LIN {X 0,Y 119.711,Z 958.893,A -85,B 0,C 180,E1 26114.773,E2 26114.773} C_VEL
LIN {X 0,Y 103.923,Z 964.098,A -85,B 0,C 180,E1 26117.575,E2 26117.575} C_VEL
LIN {X 0,Y 73.939,Z 972.907,A -85,B 0,C 180,E1 26135.275,E2 26135.275} C_VEL
LIN {X 0,Y 58.903,Z 976.31,A -85,B 0,C 180,E1 26159.176,E2 26159.176} C_VEL
LIN {X 0,Y 56.099,Z 976.57,A -85,B 0,C 180,E1 26189.998,E2 26189.998} C_VEL
LIN {X 0,Y 59.186,Z 972.492,A -85,B 0,C 180,E1 26220.657,E2 26220.657} C_VEL
LIN {X 0,Y 76.443,Z 963.091,A -85,B 0,C 180,E1 26247.029,E2 26247.029} C_VEL
LIN {X 0,Y 104.465,Z 947.144,A -85,B 0,C 180,E1 26263.142,E2 26263.142} C_VEL
LIN {X 0,Y 134.627,Z 925.946,A -85,B 0,C 180,E1 26271.712,E2 26271.712} C_VEL
LIN {X 0,Y 162.508,Z 900.972,A -85,B 0,C 180,E1 26276.579,E2 26276.579} C_VEL
LIN {X 0,Y 170.712,Z 892.031,A -85,B 0,C 180,E1 26277.998,E2 26277.998} C_VEL
LIN {X 0,Y 172.966,Z 882.755,A -85,B 0,C 180,E1 26286.219,E2 26286.219} C_VEL
LIN {X 0,Y 173.334,Z 880.134,A -85,B 0,C 180,E1 26289.984,E2 26289.984} C_VEL
LIN {X 0,Y 171.958,Z 879.719,A -85,B 0,C 180,E1 26295.218,E2 26295.218} C_VEL
LIN {X 0,Y 170.223,Z 881.343,A -85,B 0,C 180,E1 26303.461,E2 26303.461} C_VEL
LIN {X 0,Y 168.527,Z 885.017,A -85,B 0,C 180,E1 26309.922,E2 26309.922} C_VEL
LIN {X 0,Y 166.252,Z 890.112,A -85,B 0,C 180,E1 26315.225,E2 26315.225} C_VEL
LIN {X 0,Y 138.554,Z 915.597,A -85,B 0,C 180,E1 26320.326,E2 26320.326} C_VEL
LIN {X 0,Y 110.78,Z 935.517,A -85,B 0,C 180,E1 26327.957,E2 26327.957} C_VEL
LIN {X 0,Y 84.761,Z 950.496,A -85,B 0,C 180,E1 26340.688,E2 26340.688} C_VEL
LIN {X 0,Y 63.942,Z 960.925,A -85,B 0,C 180,E1 26363.225,E2 26363.225} C_VEL
LIN {X 0,Y 56.022,Z 965.379,A -85,B 0,C 180,E1 26385.628,E2 26385.628} C_VEL
LIN {X 0,Y 59.105,Z 968.135,A -85,B 0,C 180,E1 26419.994,E2 26419.994} C_VEL
LIN {X 0,Y 77.778,Z 966.879,A -85,B 0,C 180,E1 26445.956,E2 26445.956} C_VEL
LIN {X 0,Y 110.4,Z 960.103,A -85,B 0,C 180,E1 26463.301,E2 26463.301} C_VEL
LIN {X 0,Y 132.48,Z 953.174,A -85,B 0,C 180,E1 26469.432,E2 26469.432} C_VEL
LIN {X 0,Y 103.923,Z 964.098,A -85,B 0,C 180,E1 26477.575,E2 26477.575} C_VEL
LIN {X 0,Y 88.187,Z 968.35,A -85,B 0,C 180,E1 26481.478,E2 26481.478} C_VEL
LIN {X 0,Y 72.86,Z 971.58,A -85,B 0,C 180,E1 26487.114,E2 26487.114} C_VEL
LIN {X 0,Y 52.121,Z 975.608,A -85,B 0,C 180,E1 26514.614,E2 26514.614} C_VEL
LIN {X 0,Y 48.161,Z 975.76,A -85,B 0,C 180,E1 26549.998,E2 26549.998} C_VEL
LIN {X 0,Y 52.398,Z 971.472,A -85,B 0,C 180,E1 26585.166,E2 26585.166} C_VEL
LIN {X 0,Y 72.034,Z 961.958,A -85,B 0,C 180,E1 26612.291,E2 26612.291} C_VEL
LIN {X 0,Y 102.362,Z 945.563,A -85,B 0,C 180,E1 26627.605,E2 26627.605} C_VEL
LIN {X 0,Y 132.171,Z 925.212,A -85,B 0,C 180,E1 26634.962,E2 26634.962} C_VEL
LIN {X 0,Y 161.894,Z 898.969,A -85,B 0,C 180,E1 26639.462,E2 26639.462} C_VEL
LIN {X 0,Y 165.333,Z 895.412,A -85,B 0,C 180,E1 26639.958,E2 26639.958} C_VEL
LIN {X 0,Y 167.77,Z 887.011,A -85,B 0,C 180,E1 26648.352,E2 26648.352} C_VEL
LIN {X 0,Y 167.887,Z 885.942,A -85,B 0,C 180,E1 26650.312,E2 26650.312} C_VEL
LIN {X 0,Y 166.423,Z 885.651,A -85,B 0,C 180,E1 26655.737,E2 26655.737} C_VEL
LIN {X 0,Y 164.66,Z 887.179,A -85,B 0,C 180,E1 26663.589,E2 26663.589} C_VEL
LIN {X 0,Y 163.034,Z 890.313,A -85,B 0,C 180,E1 26669.203,E2 26669.203} C_VEL
LIN {X 0,Y 161.386,Z 893.294,A -85,B 0,C 180,E1 26672.698,E2 26672.698} C_VEL
LIN {X 0,Y 152.966,Z 901.547,A -85,B 0,C 180,E1 26674.291,E2 26674.291} C_VEL
LIN {X 0,Y 123.005,Z 925.698,A -85,B 0,C 180,E1 26679.938,E2 26679.938} C_VEL
LIN {X 0,Y 92.965,Z 944.319,A -85,B 0,C 180,E1 26689.514,E2 26689.514} C_VEL
LIN {X 0,Y 66.823,Z 957.209,A -85,B 0,C 180,E1 26706.828,E2 26706.828} C_VEL
LIN {X 0,Y 52.071,Z 963.832,A -85,B 0,C 180,E1 26730.002,E2 26730.002} C_VEL
LIN {X 0,Y 48.032,Z 968.202,A -85,B 0,C 180,E1 26768.931,E2 26768.931} C_VEL
LIN {X 0,Y 63.418,Z 968.657,A -85,B 0,C 180,E1 26802.143,E2 26802.143} C_VEL
LIN {X 0,Y 96.013,Z 964.023,A -85,B 0,C 180,E1 26823.196,E2 26823.196} C_VEL
LIN {X 0,Y 114.587,Z 959.44,A -85,B 0,C 180,E1 26829.148,E2 26829.148} C_VEL
LIN {X 0,Y 80.764,Z 969.716,A -85,B 0,C 180,E1 26842.03,E2 26842.03} C_VEL
LIN {X 0,Y 72.86,Z 971.58,A -85,B 0,C 180,E1 26847.114,E2 26847.114} C_VEL
LIN {X 0,Y 58.467,Z 973.826,A -85,B 0,C 180,E1 26855.615,E2 26855.615} C_VEL
LIN {X 0,Y 45.635,Z 974.913,A -85,B 0,C 180,E1 26868.941,E2 26868.941} C_VEL
LIN {X 0,Y 40.215,Z 974.944,A -85,B 0,C 180,E1 26909.997,E2 26909.997} C_VEL
LIN {X 0,Y 45.994,Z 970.426,A -85,B 0,C 180,E1 26951.006,E2 26951.006} C_VEL
LIN {X 0,Y 71.033,Z 959.531,A -85,B 0,C 180,E1 26979.966,E2 26979.966} C_VEL
LIN {X 0,Y 100.479,Z 944.235,A -85,B 0,C 180,E1 26992.068,E2 26992.068} C_VEL
LIN {X 0,Y 132.074,Z 922.944,A -85,B 0,C 180,E1 26998.663,E2 26998.663} C_VEL
LIN {X 0,Y 160.083,Z 898.33,A -85,B 0,C 180,E1 27002.382,E2 27002.382} C_VEL
LIN {X 0,Y 162.144,Z 892.536,A -85,B 0,C 180,E1 27008.644,E2 27008.644} C_VEL
LIN {X 0,Y 162.183,Z 891.558,A -85,B 0,C 180,E1 27010.679,E2 27010.679} C_VEL
LIN {X 0,Y 159.928,Z 891.844,A -85,B 0,C 180,E1 27019.343,E2 27019.343} C_VEL
LIN {X 0,Y 158.168,Z 894.158,A -85,B 0,C 180,E1 27026.512,E2 27026.512} C_VEL
LIN {X 0,Y 155.869,Z 897.582,A -85,B 0,C 180,E1 27030.772,E2 27030.772} C_VEL
LIN {X 0,Y 125.105,Z 922.932,A -85,B 0,C 180,E1 27035.494,E2 27035.494} C_VEL
LIN {X 0,Y 93.629,Z 942.489,A -85,B 0,C 180,E1 27043.511,E2 27043.511} C_VEL
LIN {X 0,Y 65.062,Z 956.148,A -85,B 0,C 180,E1 27058.545,E2 27058.545} C_VEL
LIN {X 0,Y 45.303,Z 964.232,A -85,B 0,C 180,E1 27085.116,E2 27085.116} C_VEL
LIN {X 0,Y 41.415,Z 969.099,A -85,B 0,C 180,E1 27136.784,E2 27136.784} C_VEL
LIN {X 0,Y 61.198,Z 969.344,A -85,B 0,C 180,E1 27170.523,E2 27170.523} C_VEL
LIN {X 0,Y 97.33,Z 964.29,A -85,B 0,C 180,E1 27188.989,E2 27188.989} C_VEL
LIN {X 0,Y 65.834,Z 971.78,A -85,B 0,C 180,E1 27203.524,E2 27203.524} C_VEL
LIN {X 0,Y 45.635,Z 974.913,A -85,B 0,C 180,E1 27228.941,E2 27228.941} C_VEL
LIN {X 0,Y 36.743,Z 974.992,A -85,B 0,C 180,E1 27250.159,E2 27250.159} C_VEL
LIN {X 0,Y 31.959,Z 973.487,A -85,B 0,C 180,E1 27279.171,E2 27279.171} C_VEL
LIN {X 0,Y 40.22,Z 969.374,A -85,B 0,C 180,E1 27318.619,E2 27318.619} C_VEL
LIN {X 0,Y 66.986,Z 958.913,A -85,B 0,C 180,E1 27345.601,E2 27345.601} C_VEL
LIN {X 0,Y 100.621,Z 942.076,A -85,B 0,C 180,E1 27356.978,E2 27356.978} C_VEL
LIN {X 0,Y 134.05,Z 919.516,A -85,B 0,C 180,E1 27362.481,E2 27362.481} C_VEL
LIN {X 0,Y 154.859,Z 901.45,A -85,B 0,C 180,E1 27364.846,E2 27364.846} C_VEL
LIN {X 0,Y 156.143,Z 898.412,A -85,B 0,C 180,E1 27368.288,E2 27368.288} C_VEL
LIN {X 0,Y 156.339,Z 897.044,A -85,B 0,C 180,E1 27371.083,E2 27371.083} C_VEL
LIN {X 0,Y 154.75,Z 897.004,A -85,B 0,C 180,E1 27376.959,E2 27376.959} C_VEL
LIN {X 0,Y 153.208,Z 898.276,A -85,B 0,C 180,E1 27383.147,E2 27383.147} C_VEL
LIN {X 0,Y 151.455,Z 900.693,A -85,B 0,C 180,E1 27388.014,E2 27388.014} C_VEL
LIN {X 0,Y 122.429,Z 923.851,A -85,B 0,C 180,E1 27392.072,E2 27392.072} C_VEL
LIN {X 0,Y 91.761,Z 942.438,A -85,B 0,C 180,E1 27398.636,E2 27398.636} C_VEL
LIN {X 0,Y 61.36,Z 956.339,A -85,B 0,C 180,E1 27412.063,E2 27412.063} C_VEL
LIN {X 0,Y 37.169,Z 965.222,A -85,B 0,C 180,E1 27442.856,E2 27442.856} C_VEL
LIN {X 0,Y 31.309,Z 968.568,A -85,B 0,C 180,E1 27478.818,E2 27478.818} C_VEL
LIN {X 0,Y 46.446,Z 970.459,A -85,B 0,C 180,E1 27527.092,E2 27527.092} C_VEL
LIN {X 0,Y 80.023,Z 967.951,A -85,B 0,C 180,E1 27548.91,E2 27548.91} C_VEL
LIN {X 0,Y 50.488,Z 973.087,A -85,B 0,C 180,E1 27566.272,E2 27566.272} C_VEL
LIN {X 0,Y 32.535,Z 974.518,A -85,B 0,C 180,E1 27608.614,E2 27608.614} C_VEL
LIN {X 0,Y 32.289,Z 974.094,A -85,B 0,C 180,E1 27629.997,E2 27629.997} C_VEL
LIN {X 0,Y 31.959,Z 973.487,A -85,B 0,C 180,E1 27639.171,E2 27639.171} C_VEL
LIN {X 0,Y 31.956,Z 971.586,A -85,B 0,C 180,E1 27662.601,E2 27662.601} C_VEL
LIN {X 0,Y 40.054,Z 966.811,A -85,B 0,C 180,E1 27695.217,E2 27695.217} C_VEL
LIN {X 0,Y 72.676,Z 954.478,A -85,B 0,C 180,E1 27715.255,E2 27715.255} C_VEL
LIN {X 0,Y 105.736,Z 937.275,A -85,B 0,C 180,E1 27722.569,E2 27722.569} C_VEL
LIN {X 0,Y 138.365,Z 914.337,A -85,B 0,C 180,E1 27726.394,E2 27726.394} C_VEL
LIN {X 0,Y 148.68,Z 905.586,A -85,B 0,C 180,E1 27727.21,E2 27727.21} C_VEL
LIN {X 0,Y 150.135,Z 903.774,A -85,B 0,C 180,E1 27728.542,E2 27728.542} C_VEL
LIN {X 0,Y 150.356,Z 902.432,A -85,B 0,C 180,E1 27731.53,E2 27731.53} C_VEL
LIN {X 0,Y 147.324,Z 903.497,A -85,B 0,C 180,E1 27742.802,E2 27742.802} C_VEL
LIN {X 0,Y 145.718,Z 905.164,A -85,B 0,C 180,E1 27745.71,E2 27745.71} C_VEL
LIN {X 0,Y 112.822,Z 929.64,A -85,B 0,C 180,E1 27749.614,E2 27749.614} C_VEL
LIN {X 0,Y 79.724,Z 947.662,A -85,B 0,C 180,E1 27756.446,E2 27756.446} C_VEL
LIN {X 0,Y 48.468,Z 960.086,A -85,B 0,C 180,E1 27771.491,E2 27771.491} C_VEL
LIN {X 0,Y 26.098,Z 967.262,A -85,B 0,C 180,E1 27810.004,E2 27810.004} C_VEL
LIN {X 0,Y 31.853,Z 970.838,A -85,B 0,C 180,E1 27881.359,E2 27881.359} C_VEL
LIN {X 0,Y 61.018,Z 970.628,A -85,B 0,C 180,E1 27908.402,E2 27908.402} C_VEL
LIN {X 0,Y 61.163,Z 970.689,A -85,B 0,C 180,E1 27909.277,E2 27909.277} C_VEL
LIN {X 0,Y 35.19,Z 973.51,A -85,B 0,C 180,E1 27930.941,E2 27930.941} C_VEL
LIN {X 0,Y 24.337,Z 973.195,A -85,B 0,C 180,E1 27989.995,E2 27989.995} C_VEL
LIN {X 0,Y 35.366,Z 968.304,A -85,B 0,C 180,E1 28048.575,E2 28048.575} C_VEL
LIN {X 0,Y 40.054,Z 966.811,A -85,B 0,C 180,E1 28055.217,E2 28055.217} C_VEL
LIN {X 0,Y 46.016,Z 964.52,A -85,B 0,C 180,E1 28063.199,E2 28063.199} C_VEL
LIN {X 0,Y 63.342,Z 956.829,A -85,B 0,C 180,E1 28079.399,E2 28079.399} C_VEL
LIN {X 0,Y 65.271,Z 956.031,A -85,B 0,C 180,E1 28080.019,E2 28080.019} C_VEL
LIN {X 0,Y 100.591,Z 938.959,A -85,B 0,C 180,E1 28086.367,E2 28086.367} C_VEL
LIN {X 0,Y 133.651,Z 916.81,A -85,B 0,C 180,E1 28089.355,E2 28089.355} C_VEL
LIN {X 0,Y 144.15,Z 908.185,A -85,B 0,C 180,E1 28090.179,E2 28090.179} C_VEL
LIN {X 0,Y 142.563,Z 907.744,A -85,B 0,C 180,E1 28097.705,E2 28097.705} C_VEL
LIN {X 0,Y 140.416,Z 909.376,A -85,B 0,C 180,E1 28102.97,E2 28102.97} C_VEL
LIN {X 0,Y 107.202,Z 932.703,A -85,B 0,C 180,E1 28106.187,E2 28106.187} C_VEL
LIN {X 0,Y 75.19,Z 949.25,A -85,B 0,C 180,E1 28111.469,E2 28111.469} C_VEL
LIN {X 0,Y 42.298,Z 961.373,A -85,B 0,C 180,E1 28124.481,E2 28124.481} C_VEL
LIN {X 0,Y 17.317,Z 968.386,A -85,B 0,C 180,E1 28170.007,E2 28170.007} C_VEL
LIN {X 0,Y 32.04,Z 971.828,A -85,B 0,C 180,E1 28260.217,E2 28260.217} C_VEL
LIN {X 0,Y 42.169,Z 972.094,A -85,B 0,C 180,E1 28269.553,E2 28269.553} C_VEL
LIN {X 0,Y 16.495,Z 972.674,A -85,B 0,C 180,E1 28327.215,E2 28327.215} C_VEL
LIN {X 0,Y 16.391,Z 972.293,A -85,B 0,C 180,E1 28349.993,E2 28349.993} C_VEL
LIN {X 0,Y 31.887,Z 967.221,A -85,B 0,C 180,E1 28421.159,E2 28421.159} C_VEL
LIN {X 0,Y 65.271,Z 956.031,A -85,B 0,C 180,E1 28440.019,E2 28440.019} C_VEL
LIN {X 0,Y 79.491,Z 949.248,A -85,B 0,C 180,E1 28446.128,E2 28446.128} C_VEL
LIN {X 0,Y 93.92,Z 941.499,A -85,B 0,C 180,E1 28450.39,E2 28450.39} C_VEL
LIN {X 0,Y 127.879,Z 920.126,A -85,B 0,C 180,E1 28452.538,E2 28452.538} C_VEL
LIN {X 0,Y 136.131,Z 913.817,A -85,B 0,C 180,E1 28452.903,E2 28452.903} C_VEL
LIN {X 0,Y 137.462,Z 912.657,A -85,B 0,C 180,E1 28453.417,E2 28453.417} C_VEL
LIN {X 0,Y 135.813,Z 913.036,A -85,B 0,C 180,E1 28459.412,E2 28459.412} C_VEL
LIN {X 0,Y 134.055,Z 914.378,A -85,B 0,C 180,E1 28460.104,E2 28460.104} C_VEL
LIN {X 0,Y 100.047,Z 936.867,A -85,B 0,C 180,E1 28462.509,E2 28462.509} C_VEL
LIN {X 0,Y 63.663,Z 953.883,A -85,B 0,C 180,E1 28467.257,E2 28467.257} C_VEL
LIN {X 0,Y 29.277,Z 964.672,A -85,B 0,C 180,E1 28479.369,E2 28479.369} C_VEL
LIN {X 0,Y 7.722,Z 970.149,A -85,B 0,C 180,E1 28568.263,E2 28568.263} C_VEL
LIN {X 0,Y 21.172,Z 972.047,A -85,B 0,C 180,E1 28627.608,E2 28627.608} C_VEL
LIN {X 0,Y 16.058,Z 972.08,A -85,B 0,C 180,E1 28639.974,E2 28639.974} C_VEL
LIN {X 0,Y 8.431,Z 971.381,A -85,B 0,C 180,E1 28709.987,E2 28709.987} C_VEL
LIN {X 0,Y 30.254,Z 966.123,A -85,B 0,C 180,E1 28795.944,E2 28795.944} C_VEL
LIN {X 0,Y 68.056,Z 953.688,A -85,B 0,C 180,E1 28807.554,E2 28807.554} C_VEL
LIN {X 0,Y 93.92,Z 941.499,A -85,B 0,C 180,E1 28810.39,E2 28810.39} C_VEL
LIN {X 0,Y 108.248,Z 933.006,A -85,B 0,C 180,E1 28813.505,E2 28813.505} C_VEL
LIN {X 0,Y 122.196,Z 923.511,A -85,B 0,C 180,E1 28815.958,E2 28815.958} C_VEL
LIN {X 0,Y 129.102,Z 918.581,A -85,B 0,C 180,E1 28816.078,E2 28816.078} C_VEL
LIN {X 0,Y 124.315,Z 921.857,A -85,B 0,C 180,E1 28816.988,E2 28816.988} C_VEL
LIN {X 0,Y 90.831,Z 942.024,A -85,B 0,C 180,E1 28818.318,E2 28818.318} C_VEL
LIN {X 0,Y 52.563,Z 958.116,A -85,B 0,C 180,E1 28821.092,E2 28821.092} C_VEL
LIN {X 0,Y 24.778,Z 965.851,A -85,B 0,C 180,E1 28824.015,E2 28824.015} C_VEL
LIN {X 0,Y 0.464,Z 970.462,A -85,B 0,C 180,E1 28709.757,E2 28709.757} C_VEL
LIN {X 0,Y 30.769,Z 964.938,A -85,B 0,C 180,E1 28811.24,E2 28811.24} C_VEL
LIN {X 0,Y 66.139,Z 953.616,A -85,B 0,C 180,E1 28814.152,E2 28814.152} C_VEL
LIN {X 0,Y 101.772,Z 936.397,A -85,B 0,C 180,E1 28815.471,E2 28815.471} C_VEL
LIN {X 0,Y 122.196,Z 923.511,A -85,B 0,C 180,E1 28815.958,E2 28815.958} C_VEL
LIN {X 0,Y 125.353,Z 925.139,A -85,B 0,C 180,E1 28816.04,E2 28816.04} C_VEL
LIN {X 0,Y 125.353,Z 1015.5,A -85,B 0,C 180,E1 28816.04,E2 28816.04} C_VEL
LIN {X 0,Y 125.353,Z 1015.5,A -85,B 0,C 180,E1 28816.04,E2 28816.04}

QRS_NEXT_CUT()
PTP {E1 28976.873,E2 28976.873}
PTP {X 0,Y 607.916,A -85,B 0,C 180,E1 28976.873,E2 28976.873,E3 0,E4 0,E5 0,E6 0}
QRS_SPEED_INIT()
LIN {X 0,Y 607.916,Z 1015.5,A -85,B 0,C 180,E1 28976.873,E2 28976.873,E3 0,E4 0,E5 0,E6 0} C_VEL
LIN {X 0,Y 607.916,Z 400.085,A -85,B 0,C 180,E1 28976.873,E2 28976.873} C_VEL
LIN {X 0,Y 607.916,Z 392.009,A -85,B 0,C 180,E1 28976.873,E2 28976.873} C_VEL
LIN {X 0,Y 607.891,Z 390.009,A -85,B 0,C 180,E1 28976.684,E2 28976.684} C_VEL
LIN {X 0,Y 607.87,Z 390.013,A -85,B 0,C 180,E1 28973.673,E2 28973.673} C_VEL
LIN {X 0,Y 607.89,Z 390.008,A -85,B 0,C 180,E1 28970.437,E2 28970.437} C_VEL
LIN {X 0,Y 607.892,Z 390.014,A -85,B 0,C 180,E1 28967.364,E2 28967.364} C_VEL
LIN {X 0,Y 607.887,Z 390.007,A -85,B 0,C 180,E1 28964.155,E2 28964.155} C_VEL
LIN {X 0,Y 607.914,Z 390.015,A -85,B 0,C 180,E1 28960.994,E2 28960.994} C_VEL
LIN {X 0,Y 607.883,Z 390.008,A -85,B 0,C 180,E1 28957.771,E2 28957.771} C_VEL
LIN {X 0,Y 607.906,Z 390.012,A -85,B 0,C 180,E1 28954.682,E2 28954.682} C_VEL
LIN {X 0,Y 607.888,Z 390.01,A -85,B 0,C 180,E1 28951.51,E2 28951.51} C_VEL
LIN {X 0,Y 607.904,Z 390.198,A -85,B 0,C 180,E1 28949.07,E2 28949.07} C_VEL
LIN {X 0,Y 607.917,Z 394.228,A -85,B 0,C 180,E1 28948.733,E2 28948.733} C_VEL
LIN {X 0,Y 607.919,Z 437.692,A -85,B 0,C 180,E1 28945.648,E2 28945.648} C_VEL
LIN {X 0,Y 607.909,Z 452.342,A -85,B 0,C 180,E1 28944.642,E2 28944.642} C_VEL
LIN {X 0,Y 607.915,Z 681.342,A -85,B 0,C 180,E1 28941.679,E2 28941.679} C_VEL
LIN {X 0,Y 607.916,Z 715.007,A -85,B 0,C 180,E1 28941.219,E2 28941.219} C_VEL
LIN {X 0,Y 607.906,Z 735.187,A -85,B 0,C 180,E1 28940.771,E2 28940.771} C_VEL
LIN {X 0,Y 607.911,Z 754.308,A -85,B 0,C 180,E1 28940.178,E2 28940.178} C_VEL
LIN {X 0,Y 607.909,Z 774.728,A -85,B 0,C 180,E1 28939.358,E2 28939.358} C_VEL
LIN {X 0,Y 607.917,Z 793.066,A -85,B 0,C 180,E1 28938.443,E2 28938.443} C_VEL
LIN {X 0,Y 607.916,Z 811.339,A -85,B 0,C 180,E1 28937.341,E2 28937.341} C_VEL
LIN {X 0,Y 607.914,Z 829.252,A -85,B 0,C 180,E1 28936.046,E2 28936.046} C_VEL
LIN {X 0,Y 607.917,Z 846.214,A -85,B 0,C 180,E1 28934.588,E2 28934.588} C_VEL
LIN {X 0,Y 607.909,Z 861.448,A -85,B 0,C 180,E1 28933.04,E2 28933.04} C_VEL
LIN {X 0,Y 607.918,Z 875.235,A -85,B 0,C 180,E1 28931.386,E2 28931.386} C_VEL
LIN {X 0,Y 607.914,Z 887.272,A -85,B 0,C 180,E1 28929.669,E2 28929.669} C_VEL
LIN {X 0,Y 607.905,Z 897.319,A -85,B 0,C 180,E1 28927.958,E2 28927.958} C_VEL
LIN {X 0,Y 607.901,Z 906.432,A -85,B 0,C 180,E1 28926.07,E2 28926.07} C_VEL
LIN {X 0,Y 607.9,Z 913.506,A -85,B 0,C 180,E1 28924.226,E2 28924.226} C_VEL
LIN {X 0,Y 607.899,Z 919.069,A -85,B 0,C 180,E1 28922.31,E2 28922.31} C_VEL
LIN {X 0,Y 607.9,Z 922.757,A -85,B 0,C 180,E1 28920.434,E2 28920.434} C_VEL
LIN {X 0,Y 607.9,Z 924.923,A -85,B 0,C 180,E1 28918.485,E2 28918.485} C_VEL
LIN {X 0,Y 607.902,Z 925.392,A -85,B 0,C 180,E1 28916.467,E2 28916.467} C_VEL
LIN {X 0,Y 607.907,Z 924.09,A -85,B 0,C 180,E1 28914.483,E2 28914.483} C_VEL
LIN {X 0,Y 607.914,Z 921.318,A -85,B 0,C 180,E1 28912.633,E2 28912.633} C_VEL
LIN {X 0,Y 607.918,Z 916.682,A -85,B 0,C 180,E1 28910.706,E2 28910.706} C_VEL
LIN {X 0,Y 607.909,Z 910.708,A -85,B 0,C 180,E1 28908.903,E2 28908.903} C_VEL
LIN {X 0,Y 607.9,Z 902.729,A -85,B 0,C 180,E1 28907.021,E2 28907.021} C_VEL
LIN {X 0,Y 607.903,Z 893.474,A -85,B 0,C 180,E1 28905.255,E2 28905.255} C_VEL
LIN {X 0,Y 607.907,Z 882.395,A -85,B 0,C 180,E1 28903.504,E2 28903.504} C_VEL
LIN {X 0,Y 607.913,Z 869.197,A -85,B 0,C 180,E1 28901.765,E2 28901.765} C_VEL
LIN {X 0,Y 607.914,Z 854.508,A -85,B 0,C 180,E1 28900.134,E2 28900.134} C_VEL
LIN {X 0,Y 607.916,Z 838.768,A -85,B 0,C 180,E1 28898.653,E2 28898.653} C_VEL
LIN {X 0,Y 607.915,Z 822.476,A -85,B 0,C 180,E1 28897.352,E2 28897.352} C_VEL
LIN {X 0,Y 607.918,Z 805.221,A -85,B 0,C 180,E1 28896.182,E2 28896.182} C_VEL
LIN {X 0,Y 607.916,Z 786.897,A -85,B 0,C 180,E1 28895.141,E2 28895.141} C_VEL
LIN {X 0,Y 607.917,Z 768.828,A -85,B 0,C 180,E1 28894.29,E2 28894.29} C_VEL
LIN {X 0,Y 607.916,Z 749.3,A -85,B 0,C 180,E1 28893.558,E2 28893.558} C_VEL
LIN {X 0,Y 607.908,Z 730.169,A -85,B 0,C 180,E1 28893.015,E2 28893.015} C_VEL
LIN {X 0,Y 607.912,Z 709.347,A -85,B 0,C 180,E1 28892.602,E2 28892.602} C_VEL
LIN {X 0,Y 607.91,Z 453.431,A -85,B 0,C 180,E1 28889.291,E2 28889.291} C_VEL
LIN {X 0,Y 607.904,Z 451.144,A -85,B 0,C 180,E1 28889.197,E2 28889.197} C_VEL
LIN {X 0,Y 607.918,Z 406.873,A -85,B 0,C 180,E1 28886.084,E2 28886.084} C_VEL
LIN {X 0,Y 607.905,Z 390.386,A -85,B 0,C 180,E1 28884.879,E2 28884.879} C_VEL
LIN {X 0,Y 607.885,Z 390.007,A -85,B 0,C 180,E1 28884.334,E2 28884.334} C_VEL
LIN {X 0,Y 607.904,Z 390.011,A -85,B 0,C 180,E1 28881.2,E2 28881.2} C_VEL
LIN {X 0,Y 607.888,Z 390.007,A -85,B 0,C 180,E1 28878.037,E2 28878.037} C_VEL
LIN {X 0,Y 607.906,Z 390.012,A -85,B 0,C 180,E1 28874.901,E2 28874.901} C_VEL
LIN {X 0,Y 607.89,Z 390.007,A -85,B 0,C 180,E1 28871.788,E2 28871.788} C_VEL
LIN {X 0,Y 607.909,Z 390.013,A -85,B 0,C 180,E1 28868.581,E2 28868.581} C_VEL
LIN {X 0,Y 607.905,Z 390.004,A -85,B 0,C 180,E1 28865.305,E2 28865.305} C_VEL
LIN {X 0,Y 607.905,Z 390.013,A -85,B 0,C 180,E1 28862.036,E2 28862.036} C_VEL
LIN {X 0,Y 607.908,Z 390.005,A -85,B 0,C 180,E1 28858.79,E2 28858.79} C_VEL
LIN {X 0,Y 607.895,Z 390.011,A -85,B 0,C 180,E1 28855.655,E2 28855.655} C_VEL
LIN {X 0,Y 607.904,Z 390.006,A -85,B 0,C 180,E1 28852.513,E2 28852.513} C_VEL
LIN {X 0,Y 607.892,Z 390.01,A -85,B 0,C 180,E1 28849.311,E2 28849.311} C_VEL
LIN {X 0,Y 607.9,Z 390.007,A -85,B 0,C 180,E1 28846.175,E2 28846.175} C_VEL
LIN {X 0,Y 607.892,Z 390.009,A -85,B 0,C 180,E1 28843.047,E2 28843.047} C_VEL
LIN {X 0,Y 607.898,Z 390.008,A -85,B 0,C 180,E1 28839.901,E2 28839.901} C_VEL
LIN {X 0,Y 607.892,Z 390.008,A -85,B 0,C 180,E1 28836.772,E2 28836.772} C_VEL
LIN {X 0,Y 607.896,Z 390.009,A -85,B 0,C 180,E1 28833.662,E2 28833.662} C_VEL
LIN {X 0,Y 607.893,Z 390.009,A -85,B 0,C 180,E1 28830.547,E2 28830.547} C_VEL
LIN {X 0,Y 607.897,Z 390.009,A -85,B 0,C 180,E1 28827.422,E2 28827.422} C_VEL
LIN {X 0,Y 607.893,Z 390.008,A -85,B 0,C 180,E1 28824.28,E2 28824.28} C_VEL
LIN {X 0,Y 607.897,Z 390.01,A -85,B 0,C 180,E1 28821.113,E2 28821.113} C_VEL
LIN {X 0,Y 607.896,Z 390.008,A -85,B 0,C 180,E1 28818.013,E2 28818.013} C_VEL
LIN {X 0,Y 607.896,Z 390.01,A -85,B 0,C 180,E1 28814.868,E2 28814.868} C_VEL
LIN {X 0,Y 607.9,Z 390.006,A -85,B 0,C 180,E1 28811.672,E2 28811.672} C_VEL
LIN {X 0,Y 607.901,Z 390.011,A -85,B 0,C 180,E1 28808.513,E2 28808.513} C_VEL
LIN {X 0,Y 607.911,Z 390.004,A -85,B 0,C 180,E1 28805.285,E2 28805.285} C_VEL
LIN {X 0,Y 607.912,Z 390.015,A -85,B 0,C 180,E1 28801.98,E2 28801.98} C_VEL
LIN {X 0,Y 607.899,Z 390.006,A -85,B 0,C 180,E1 28798.681,E2 28798.681} C_VEL
LIN {X 0,Y 607.9,Z 390.011,A -85,B 0,C 180,E1 28795.472,E2 28795.472} C_VEL
LIN {X 0,Y 607.893,Z 390.007,A -85,B 0,C 180,E1 28792.344,E2 28792.344} C_VEL
LIN {X 0,Y 607.899,Z 390.01,A -85,B 0,C 180,E1 28789.193,E2 28789.193} C_VEL
LIN {X 0,Y 607.892,Z 390.007,A -85,B 0,C 180,E1 28786.105,E2 28786.105} C_VEL
LIN {X 0,Y 607.9,Z 390.01,A -85,B 0,C 180,E1 28782.976,E2 28782.976} C_VEL
LIN {X 0,Y 607.891,Z 390.007,A -85,B 0,C 180,E1 28779.894,E2 28779.894} C_VEL
LIN {X 0,Y 607.901,Z 390.01,A -85,B 0,C 180,E1 28776.75,E2 28776.75} C_VEL
LIN {X 0,Y 607.889,Z 390.008,A -85,B 0,C 180,E1 28773.635,E2 28773.635} C_VEL
LIN {X 0,Y 607.901,Z 390.01,A -85,B 0,C 180,E1 28770.542,E2 28770.542} C_VEL
LIN {X 0,Y 607.889,Z 390.007,A -85,B 0,C 180,E1 28767.463,E2 28767.463} C_VEL
LIN {X 0,Y 607.903,Z 390.01,A -85,B 0,C 180,E1 28764.343,E2 28764.343} C_VEL
LIN {X 0,Y 607.887,Z 390.008,A -85,B 0,C 180,E1 28761.195,E2 28761.195} C_VEL
LIN {X 0,Y 607.903,Z 390.01,A -85,B 0,C 180,E1 28758.105,E2 28758.105} C_VEL
LIN {X 0,Y 607.887,Z 390.008,A -85,B 0,C 180,E1 28754.987,E2 28754.987} C_VEL
LIN {X 0,Y 607.902,Z 390.01,A -85,B 0,C 180,E1 28751.897,E2 28751.897} C_VEL
LIN {X 0,Y 607.886,Z 390.008,A -85,B 0,C 180,E1 28748.773,E2 28748.773} C_VEL
LIN {X 0,Y 607.899,Z 390.272,A -85,B 0,C 180,E1 28746.232,E2 28746.232} C_VEL
LIN {X 0,Y 607.915,Z 394.031,A -85,B 0,C 180,E1 28745.958,E2 28745.958} C_VEL
LIN {X 0,Y 607.913,Z 445.359,A -85,B 0,C 180,E1 28742.929,E2 28742.929} C_VEL
LIN {X 0,Y 607.903,Z 455.392,A -85,B 0,C 180,E1 28742.37,E2 28742.37} C_VEL
LIN {X 0,Y 607.916,Z 672.013,A -85,B 0,C 180,E1 28739.445,E2 28739.445} C_VEL
LIN {X 0,Y 607.899,Z 760.574,A -85,B 0,C 180,E1 28738.249,E2 28738.249} C_VEL
LIN {X 0,Y 607.906,Z 781.2,A -85,B 0,C 180,E1 28737.806,E2 28737.806} C_VEL
LIN {X 0,Y 607.908,Z 801.762,A -85,B 0,C 180,E1 28737.211,E2 28737.211} C_VEL
LIN {X 0,Y 607.904,Z 822.538,A -85,B 0,C 180,E1 28736.419,E2 28736.419} C_VEL
LIN {X 0,Y 607.918,Z 843.715,A -85,B 0,C 180,E1 28735.423,E2 28735.423} C_VEL
LIN {X 0,Y 607.916,Z 863.098,A -85,B 0,C 180,E1 28734.332,E2 28734.332} C_VEL
LIN {X 0,Y 607.915,Z 881.539,A -85,B 0,C 180,E1 28733.097,E2 28733.097} C_VEL
LIN {X 0,Y 607.911,Z 899.771,A -85,B 0,C 180,E1 28731.678,E2 28731.678} C_VEL
LIN {X 0,Y 607.913,Z 916.635,A -85,B 0,C 180,E1 28730.157,E2 28730.157} C_VEL
LIN {X 0,Y 607.918,Z 932.451,A -85,B 0,C 180,E1 28728.509,E2 28728.509} C_VEL
LIN {X 0,Y 607.916,Z 946.401,A -85,B 0,C 180,E1 28726.818,E2 28726.818} C_VEL
LIN {X 0,Y 607.919,Z 958.89,A -85,B 0,C 180,E1 28725.064,E2 28725.064} C_VEL
LIN {X 0,Y 607.917,Z 970.422,A -85,B 0,C 180,E1 28723.176,E2 28723.176} C_VEL
LIN {X 0,Y 607.903,Z 980.052,A -85,B 0,C 180,E1 28721.289,E2 28721.289} C_VEL
LIN {X 0,Y 607.896,Z 988.388,A -85,B 0,C 180,E1 28719.296,E2 28719.296} C_VEL
LIN {X 0,Y 607.891,Z 994.96,A -85,B 0,C 180,E1 28717.339,E2 28717.339} C_VEL
LIN {X 0,Y 607.9,Z 999.805,A -85,B 0,C 180,E1 28715.381,E2 28715.381} C_VEL
LIN {X 0,Y 607.913,Z 1003.346,A -85,B 0,C 180,E1 28713.29,E2 28713.29} C_VEL
LIN {X 0,Y 607.911,Z 1005.209,A -85,B 0,C 180,E1 28711.227,E2 28711.227} C_VEL
LIN {X 0,Y 607.894,Z 1005.329,A -85,B 0,C 180,E1 28709.248,E2 28709.248} C_VEL
LIN {X 0,Y 607.89,Z 1003.898,A -85,B 0,C 180,E1 28707.174,E2 28707.174} C_VEL
LIN {X 0,Y 607.901,Z 1001.148,A -85,B 0,C 180,E1 28705.285,E2 28705.285} C_VEL
LIN {X 0,Y 607.916,Z 996.658,A -85,B 0,C 180,E1 28703.296,E2 28703.296} C_VEL
LIN {X 0,Y 607.908,Z 990.6,A -85,B 0,C 180,E1 28701.299,E2 28701.299} C_VEL
LIN {X 0,Y 607.908,Z 983.074,A -85,B 0,C 180,E1 28699.387,E2 28699.387} C_VEL
LIN {X 0,Y 607.909,Z 973.339,A -85,B 0,C 180,E1 28697.367,E2 28697.367} C_VEL
LIN {X 0,Y 607.916,Z 962.761,A -85,B 0,C 180,E1 28695.525,E2 28695.525} C_VEL
LIN {X 0,Y 607.913,Z 950.052,A -85,B 0,C 180,E1 28693.668,E2 28693.668} C_VEL
LIN {X 0,Y 607.905,Z 935.888,A -85,B 0,C 180,E1 28691.892,E2 28691.892} C_VEL
LIN {X 0,Y 607.909,Z 920.092,A -85,B 0,C 180,E1 28690.185,E2 28690.185} C_VEL
LIN {X 0,Y 607.914,Z 903.529,A -85,B 0,C 180,E1 28688.638,E2 28688.638} C_VEL
LIN {X 0,Y 607.916,Z 885.835,A -85,B 0,C 180,E1 28687.214,E2 28687.214} C_VEL
LIN {X 0,Y 607.915,Z 867.977,A -85,B 0,C 180,E1 28685.982,E2 28685.982} C_VEL
LIN {X 0,Y 607.918,Z 848.77,A -85,B 0,C 180,E1 28684.842,E2 28684.842} C_VEL
LIN {X 0,Y 607.899,Z 829.889,A -85,B 0,C 180,E1 28683.902,E2 28683.902} C_VEL
LIN {X 0,Y 607.916,Z 809.129,A -85,B 0,C 180,E1 28683.055,E2 28683.055} C_VEL
LIN {X 0,Y 607.914,Z 789.266,A -85,B 0,C 180,E1 28682.404,E2 28682.404} C_VEL
LIN {X 0,Y 607.898,Z 769.076,A -85,B 0,C 180,E1 28681.916,E2 28681.916} C_VEL
LIN {X 0,Y 607.908,Z 747.682,A -85,B 0,C 180,E1 28681.555,E2 28681.555} C_VEL
LIN {X 0,Y 607.91,Z 522.734,A -85,B 0,C 180,E1 28678.551,E2 28678.551} C_VEL
LIN {X 0,Y 607.903,Z 454.694,A -85,B 0,C 180,E1 28677.607,E2 28677.607} C_VEL
LIN {X 0,Y 607.918,Z 404.419,A -85,B 0,C 180,E1 28674.665,E2 28674.665} C_VEL
LIN {X 0,Y 607.903,Z 390.536,A -85,B 0,C 180,E1 28673.813,E2 28673.813} C_VEL
LIN {X 0,Y 607.889,Z 390.021,A -85,B 0,C 180,E1 28673.579,E2 28673.579} C_VEL
LIN {X 0,Y 607.909,Z 390.007,A -85,B 0,C 180,E1 28670.471,E2 28670.471} C_VEL
LIN {X 0,Y 607.877,Z 390.011,A -85,B 0,C 180,E1 28667.327,E2 28667.327} C_VEL
LIN {X 0,Y 607.91,Z 390.01,A -85,B 0,C 180,E1 28664.188,E2 28664.188} C_VEL
LIN {X 0,Y 607.869,Z 390.011,A -85,B 0,C 180,E1 28661.124,E2 28661.124} C_VEL
LIN {X 0,Y 607.914,Z 390.011,A -85,B 0,C 180,E1 28658.023,E2 28658.023} C_VEL
LIN {X 0,Y 607.858,Z 390.011,A -85,B 0,C 180,E1 28654.919,E2 28654.919} C_VEL
LIN {X 0,Y 607.915,Z 390.014,A -85,B 0,C 180,E1 28651.756,E2 28651.756} C_VEL
LIN {X 0,Y 607.849,Z 390.012,A -85,B 0,C 180,E1 28648.756,E2 28648.756} C_VEL
LIN {X 0,Y 607.918,Z 390.015,A -85,B 0,C 180,E1 28645.63,E2 28645.63} C_VEL
LIN {X 0,Y 607.839,Z 390.013,A -85,B 0,C 180,E1 28642.638,E2 28642.638} C_VEL
LIN {X 0,Y 607.914,Z 390.015,A -85,B 0,C 180,E1 28639.547,E2 28639.547} C_VEL
LIN {X 0,Y 607.827,Z 390.015,A -85,B 0,C 180,E1 28636.533,E2 28636.533} C_VEL
LIN {X 0,Y 607.898,Z 390.015,A -85,B 0,C 180,E1 28633.591,E2 28633.591} C_VEL
LIN {X 0,Y 607.831,Z 390.014,A -85,B 0,C 180,E1 28630.52,E2 28630.52} C_VEL
LIN {X 0,Y 607.878,Z 390.014,A -85,B 0,C 180,E1 28627.656,E2 28627.656} C_VEL
LIN {X 0,Y 607.849,Z 390.012,A -85,B 0,C 180,E1 28624.528,E2 28624.528} C_VEL
LIN {X 0,Y 607.869,Z 390.014,A -85,B 0,C 180,E1 28621.696,E2 28621.696} C_VEL
LIN {X 0,Y 607.866,Z 390.01,A -85,B 0,C 180,E1 28618.492,E2 28618.492} C_VEL
LIN {X 0,Y 607.891,Z 390.009,A -85,B 0,C 180,E1 28616.684,E2 28616.684} C_VEL
LIN {X 0,Y 606.84,Z 390.14,A -85,B 0,C 180,E1 28615.958,E2 28615.958} C_VEL
LIN {X 0,Y 600.436,Z 390.939,A -85,B 0,C 180,E1 28613.921,E2 28613.921} C_VEL
LIN {X 0,Y 599.956,Z 391.003,A -85,B 0,C 180,E1 28613.391,E2 28613.391} C_VEL
LIN {X 0,Y 599.935,Z 390.998,A -85,B 0,C 180,E1 28610.212,E2 28610.212} C_VEL
LIN {X 0,Y 599.974,Z 391.004,A -85,B 0,C 180,E1 28607.096,E2 28607.096} C_VEL
LIN {X 0,Y 599.938,Z 390.998,A -85,B 0,C 180,E1 28603.939,E2 28603.939} C_VEL
LIN {X 0,Y 599.971,Z 391.001,A -85,B 0,C 180,E1 28600.834,E2 28600.834} C_VEL
LIN {X 0,Y 599.943,Z 390.997,A -85,B 0,C 180,E1 28597.652,E2 28597.652} C_VEL
LIN {X 0,Y 599.966,Z 390.999,A -85,B 0,C 180,E1 28594.534,E2 28594.534} C_VEL
LIN {X 0,Y 599.95,Z 391.001,A -85,B 0,C 180,E1 28591.425,E2 28591.425} C_VEL
LIN {X 0,Y 599.991,Z 391.268,A -85,B 0,C 180,E1 28589.451,E2 28589.451} C_VEL
LIN {X 0,Y 600.749,Z 394.183,A -85,B 0,C 180,E1 28589.161,E2 28589.161} C_VEL
LIN {X 0,Y 600.607,Z 437.56,A -85,B 0,C 180,E1 28586.04,E2 28586.04} C_VEL
LIN {X 0,Y 600.657,Z 452.847,A -85,B 0,C 180,E1 28584.993,E2 28584.993} C_VEL
LIN {X 0,Y 600.684,Z 617.803,A -85,B 0,C 180,E1 28582.821,E2 28582.821} C_VEL
LIN {X 0,Y 600.614,Z 714.338,A -85,B 0,C 180,E1 28581.546,E2 28581.546} C_VEL
LIN {X 0,Y 600.558,Z 734.765,A -85,B 0,C 180,E1 28581.091,E2 28581.091} C_VEL
LIN {X 0,Y 600.502,Z 753.729,A -85,B 0,C 180,E1 28580.502,E2 28580.502} C_VEL
LIN {X 0,Y 600.427,Z 772.626,A -85,B 0,C 180,E1 28579.75,E2 28579.75} C_VEL
LIN {X 0,Y 600.362,Z 791.336,A -85,B 0,C 180,E1 28578.826,E2 28578.826} C_VEL
LIN {X 0,Y 600.284,Z 810.203,A -85,B 0,C 180,E1 28577.688,E2 28577.688} C_VEL
LIN {X 0,Y 600.204,Z 827.508,A -85,B 0,C 180,E1 28576.435,E2 28576.435} C_VEL
LIN {X 0,Y 600.126,Z 843.684,A -85,B 0,C 180,E1 28575.055,E2 28575.055} C_VEL
LIN {X 0,Y 600.069,Z 858.753,A -85,B 0,C 180,E1 28573.546,E2 28573.546} C_VEL
LIN {X 0,Y 600.011,Z 872.519,A -85,B 0,C 180,E1 28571.926,E2 28571.926} C_VEL
LIN {X 0,Y 599.968,Z 885.206,A -85,B 0,C 180,E1 28570.157,E2 28570.157} C_VEL
LIN {X 0,Y 599.942,Z 895.862,A -85,B 0,C 180,E1 28568.38,E2 28568.38} C_VEL
LIN {X 0,Y 599.927,Z 904.924,A -85,B 0,C 180,E1 28566.551,E2 28566.551} C_VEL
LIN {X 0,Y 599.923,Z 912.488,A -85,B 0,C 180,E1 28564.63,E2 28564.63} C_VEL
LIN {X 0,Y 599.919,Z 917.987,A -85,B 0,C 180,E1 28562.793,E2 28562.793} C_VEL
LIN {X 0,Y 599.916,Z 922.277,A -85,B 0,C 180,E1 28560.771,E2 28560.771} C_VEL
LIN {X 0,Y 599.912,Z 924.749,A -85,B 0,C 180,E1 28558.756,E2 28558.756} C_VEL
LIN {X 0,Y 599.913,Z 925.481,A -85,B 0,C 180,E1 28556.848,E2 28556.848} C_VEL
LIN {X 0,Y 599.916,Z 924.522,A -85,B 0,C 180,E1 28554.831,E2 28554.831} C_VEL
LIN {X 0,Y 599.917,Z 921.765,A -85,B 0,C 180,E1 28552.829,E2 28552.829} C_VEL
LIN {X 0,Y 599.916,Z 917.396,A -85,B 0,C 180,E1 28550.893,E2 28550.893} C_VEL
LIN {X 0,Y 599.918,Z 911.323,A -85,B 0,C 180,E1 28548.963,E2 28548.963} C_VEL
LIN {X 0,Y 599.923,Z 904,A -85,B 0,C 180,E1 28547.155,E2 28547.155} C_VEL
LIN {X 0,Y 599.942,Z 894.448,A -85,B 0,C 180,E1 28545.265,E2 28545.265} C_VEL
LIN {X 0,Y 599.97,Z 883.49,A -85,B 0,C 180,E1 28543.49,E2 28543.49} C_VEL
LIN {X 0,Y 600.019,Z 871.269,A -85,B 0,C 180,E1 28541.825,E2 28541.825} C_VEL
LIN {X 0,Y 600.071,Z 857.858,A -85,B 0,C 180,E1 28540.268,E2 28540.268} C_VEL
LIN {X 0,Y 600.131,Z 842.182,A -85,B 0,C 180,E1 28538.718,E2 28538.718} C_VEL
LIN {X 0,Y 600.206,Z 825.476,A -85,B 0,C 180,E1 28537.319,E2 28537.319} C_VEL
LIN {X 0,Y 600.291,Z 807.905,A -85,B 0,C 180,E1 28536.076,E2 28536.076} C_VEL
LIN {X 0,Y 600.374,Z 790.021,A -85,B 0,C 180,E1 28535.014,E2 28535.014} C_VEL
LIN {X 0,Y 600.438,Z 770.836,A -85,B 0,C 180,E1 28534.078,E2 28534.078} C_VEL
LIN {X 0,Y 600.511,Z 751.093,A -85,B 0,C 180,E1 28533.315,E2 28533.315} C_VEL
LIN {X 0,Y 600.564,Z 731.085,A -85,B 0,C 180,E1 28532.726,E2 28532.726} C_VEL
LIN {X 0,Y 600.616,Z 710.383,A -85,B 0,C 180,E1 28532.303,E2 28532.303} C_VEL
LIN {X 0,Y 600.821,Z 454.166,A -85,B 0,C 180,E1 28528.946,E2 28528.946} C_VEL
LIN {X 0,Y 600.549,Z 451.544,A -85,B 0,C 180,E1 28528.853,E2 28528.853} C_VEL
LIN {X 0,Y 600.709,Z 407.289,A -85,B 0,C 180,E1 28525.703,E2 28525.703} C_VEL
LIN {X 0,Y 600.525,Z 393.145,A -85,B 0,C 180,E1 28524.659,E2 28524.659} C_VEL
LIN {X 0,Y 599.96,Z 391.101,A -85,B 0,C 180,E1 28524.415,E2 28524.415} C_VEL
LIN {X 0,Y 599.965,Z 391,A -85,B 0,C 180,E1 28521.275,E2 28521.275} C_VEL
LIN {X 0,Y 599.947,Z 390.997,A -85,B 0,C 180,E1 28518.169,E2 28518.169} C_VEL
LIN {X 0,Y 599.964,Z 390.999,A -85,B 0,C 180,E1 28515.028,E2 28515.028} C_VEL
LIN {X 0,Y 599.948,Z 390.997,A -85,B 0,C 180,E1 28511.94,E2 28511.94} C_VEL
LIN {X 0,Y 599.964,Z 390.999,A -85,B 0,C 180,E1 28508.798,E2 28508.798} C_VEL
LIN {X 0,Y 599.953,Z 390.996,A -85,B 0,C 180,E1 28505.586,E2 28505.586} C_VEL
LIN {X 0,Y 599.968,Z 391.001,A -85,B 0,C 180,E1 28502.399,E2 28502.399} C_VEL
LIN {X 0,Y 599.967,Z 390.993,A -85,B 0,C 180,E1 28499.116,E2 28499.116} C_VEL
LIN {X 0,Y 599.962,Z 391.001,A -85,B 0,C 180,E1 28495.752,E2 28495.752} C_VEL
LIN {X 0,Y 599.966,Z 390.995,A -85,B 0,C 180,E1 28492.533,E2 28492.533} C_VEL
LIN {X 0,Y 599.953,Z 390.999,A -85,B 0,C 180,E1 28489.314,E2 28489.314} C_VEL
LIN {X 0,Y 599.961,Z 390.995,A -85,B 0,C 180,E1 28486.188,E2 28486.188} C_VEL
LIN {X 0,Y 599.954,Z 390.999,A -85,B 0,C 180,E1 28483.102,E2 28483.102} C_VEL
LIN {X 0,Y 599.96,Z 390.996,A -85,B 0,C 180,E1 28479.949,E2 28479.949} C_VEL
LIN {X 0,Y 599.953,Z 390.997,A -85,B 0,C 180,E1 28476.748,E2 28476.748} C_VEL
LIN {X 0,Y 599.959,Z 390.999,A -85,B 0,C 180,E1 28473.563,E2 28473.563} C_VEL
LIN {X 0,Y 599.956,Z 390.996,A -85,B 0,C 180,E1 28470.44,E2 28470.44} C_VEL
LIN {X 0,Y 599.96,Z 391,A -85,B 0,C 180,E1 28467.278,E2 28467.278} C_VEL
LIN {X 0,Y 599.959,Z 390.995,A -85,B 0,C 180,E1 28464.099,E2 28464.099} C_VEL
LIN {X 0,Y 599.965,Z 391.001,A -85,B 0,C 180,E1 28460.894,E2 28460.894} C_VEL
LIN {X 0,Y 599.973,Z 390.993,A -85,B 0,C 180,E1 28457.556,E2 28457.556} C_VEL
LIN {X 0,Y 599.966,Z 391.001,A -85,B 0,C 180,E1 28454.279,E2 28454.279} C_VEL
LIN {X 0,Y 599.959,Z 390.995,A -85,B 0,C 180,E1 28451.05,E2 28451.05} C_VEL
LIN {X 0,Y 599.959,Z 390.999,A -85,B 0,C 180,E1 28447.855,E2 28447.855} C_VEL
LIN {X 0,Y 599.955,Z 390.997,A -85,B 0,C 180,E1 28444.684,E2 28444.684} C_VEL
LIN {X 0,Y 599.959,Z 390.998,A -85,B 0,C 180,E1 28441.528,E2 28441.528} C_VEL
LIN {X 0,Y 599.955,Z 390.998,A -85,B 0,C 180,E1 28438.377,E2 28438.377} C_VEL
LIN {X 0,Y 599.96,Z 390.997,A -85,B 0,C 180,E1 28435.22,E2 28435.22} C_VEL
LIN {X 0,Y 599.955,Z 390.998,A -85,B 0,C 180,E1 28432.049,E2 28432.049} C_VEL
LIN {X 0,Y 599.966,Z 390.994,A -85,B 0,C 180,E1 28428.854,E2 28428.854} C_VEL
LIN {X 0,Y 599.965,Z 391.002,A -85,B 0,C 180,E1 28425.623,E2 28425.623} C_VEL
LIN {X 0,Y 599.966,Z 390.993,A -85,B 0,C 180,E1 28422.244,E2 28422.244} C_VEL
LIN {X 0,Y 599.968,Z 391.001,A -85,B 0,C 180,E1 28419.004,E2 28419.004} C_VEL
LIN {X 0,Y 599.952,Z 390.996,A -85,B 0,C 180,E1 28415.797,E2 28415.797} C_VEL
LIN {X 0,Y 599.963,Z 390.999,A -85,B 0,C 180,E1 28412.616,E2 28412.616} C_VEL
LIN {X 0,Y 599.95,Z 390.998,A -85,B 0,C 180,E1 28409.449,E2 28409.449} C_VEL
LIN {X 0,Y 599.963,Z 390.997,A -85,B 0,C 180,E1 28406.264,E2 28406.264} C_VEL
LIN {X 0,Y 599.95,Z 390.999,A -85,B 0,C 180,E1 28403.127,E2 28403.127} C_VEL
LIN {X 0,Y 599.967,Z 390.995,A -85,B 0,C 180,E1 28399.902,E2 28399.902} C_VEL
LIN {X 0,Y 599.952,Z 391.001,A -85,B 0,C 180,E1 28396.744,E2 28396.744} C_VEL
LIN {X 0,Y 599.977,Z 390.993,A -85,B 0,C 180,E1 28393.494,E2 28393.494} C_VEL
LIN {X 0,Y 599.97,Z 391.004,A -85,B 0,C 180,E1 28390.162,E2 28390.162} C_VEL
LIN {X 0,Y 599.959,Z 391.049,A -85,B 0,C 180,E1 28386.868,E2 28386.868} C_VEL
LIN {X 0,Y 600.034,Z 391.535,A -85,B 0,C 180,E1 28386.677,E2 28386.677} C_VEL
LIN {X 0,Y 601.105,Z 394.791,A -85,B 0,C 180,E1 28386.383,E2 28386.383} C_VEL
LIN {X 0,Y 600.926,Z 445.429,A -85,B 0,C 180,E1 28383.358,E2 28383.358} C_VEL
LIN {X 0,Y 601.015,Z 455.728,A -85,B 0,C 180,E1 28382.781,E2 28382.781} C_VEL
LIN {X 0,Y 600.976,Z 628.754,A -85,B 0,C 180,E1 28380.405,E2 28380.405} C_VEL
LIN {X 0,Y 600.842,Z 761.002,A -85,B 0,C 180,E1 28378.604,E2 28378.604} C_VEL
LIN {X 0,Y 600.787,Z 781.966,A -85,B 0,C 180,E1 28378.145,E2 28378.145} C_VEL
LIN {X 0,Y 600.714,Z 802.505,A -85,B 0,C 180,E1 28377.537,E2 28377.537} C_VEL
LIN {X 0,Y 600.636,Z 822.541,A -85,B 0,C 180,E1 28376.764,E2 28376.764} C_VEL
LIN {X 0,Y 600.539,Z 843.718,A -85,B 0,C 180,E1 28375.758,E2 28375.758} C_VEL
LIN {X 0,Y 600.445,Z 863.085,A -85,B 0,C 180,E1 28374.655,E2 28374.655} C_VEL
LIN {X 0,Y 600.354,Z 881.419,A -85,B 0,C 180,E1 28373.414,E2 28373.414} C_VEL
LIN {X 0,Y 600.25,Z 899.254,A -85,B 0,C 180,E1 28372.013,E2 28372.013} C_VEL
LIN {X 0,Y 600.16,Z 916.128,A -85,B 0,C 180,E1 28370.48,E2 28370.48} C_VEL
LIN {X 0,Y 600.109,Z 931.646,A -85,B 0,C 180,E1 28368.852,E2 28368.852} C_VEL
LIN {X 0,Y 600.041,Z 945.547,A -85,B 0,C 180,E1 28367.155,E2 28367.155} C_VEL
LIN {X 0,Y 599.989,Z 958.892,A -85,B 0,C 180,E1 28365.268,E2 28365.268} C_VEL
LIN {X 0,Y 599.952,Z 970.202,A -85,B 0,C 180,E1 28363.396,E2 28363.396} C_VEL
LIN {X 0,Y 599.925,Z 979.847,A -85,B 0,C 180,E1 28361.484,E2 28361.484} C_VEL
LIN {X 0,Y 599.905,Z 988.102,A -85,B 0,C 180,E1 28359.499,E2 28359.499} C_VEL
LIN {X 0,Y 599.903,Z 994.578,A -85,B 0,C 180,E1 28357.568,E2 28357.568} C_VEL
LIN {X 0,Y 599.911,Z 999.599,A -85,B 0,C 180,E1 28355.549,E2 28355.549} C_VEL
LIN {X 0,Y 599.914,Z 1003.22,A -85,B 0,C 180,E1 28353.442,E2 28353.442} C_VEL
LIN {X 0,Y 599.901,Z 1005.079,A -85,B 0,C 180,E1 28351.435,E2 28351.435} C_VEL
LIN {X 0,Y 599.891,Z 1005.373,A -85,B 0,C 180,E1 28349.429,E2 28349.429} C_VEL
LIN {X 0,Y 599.896,Z 1004.234,A -85,B 0,C 180,E1 28347.423,E2 28347.423} C_VEL
LIN {X 0,Y 599.909,Z 1001.465,A -85,B 0,C 180,E1 28345.414,E2 28345.414} C_VEL
LIN {X 0,Y 599.92,Z 996.912,A -85,B 0,C 180,E1 28343.303,E2 28343.303} C_VEL
LIN {X 0,Y 599.92,Z 990.79,A -85,B 0,C 180,E1 28341.234,E2 28341.234} C_VEL
LIN {X 0,Y 599.927,Z 983.074,A -85,B 0,C 180,E1 28339.244,E2 28339.244} C_VEL
LIN {X 0,Y 599.949,Z 973.34,A -85,B 0,C 180,E1 28337.196,E2 28337.196} C_VEL
LIN {X 0,Y 599.988,Z 962.76,A -85,B 0,C 180,E1 28335.33,E2 28335.33} C_VEL
LIN {X 0,Y 600.025,Z 950.053,A -85,B 0,C 180,E1 28333.447,E2 28333.447} C_VEL
LIN {X 0,Y 600.075,Z 935.889,A -85,B 0,C 180,E1 28331.647,E2 28331.647} C_VEL
LIN {X 0,Y 600.155,Z 920.222,A -85,B 0,C 180,E1 28329.931,E2 28329.931} C_VEL
LIN {X 0,Y 600.24,Z 904.134,A -85,B 0,C 180,E1 28328.402,E2 28328.402} C_VEL
LIN {X 0,Y 600.32,Z 885.835,A -85,B 0,C 180,E1 28326.909,E2 28326.909} C_VEL
LIN {X 0,Y 600.421,Z 867.177,A -85,B 0,C 180,E1 28325.611,E2 28325.611} C_VEL
LIN {X 0,Y 600.533,Z 846.786,A -85,B 0,C 180,E1 28324.405,E2 28324.405} C_VEL
LIN {X 0,Y 600.599,Z 827.613,A -85,B 0,C 180,E1 28323.452,E2 28323.452} C_VEL
LIN {X 0,Y 600.701,Z 807.046,A -85,B 0,C 180,E1 28322.628,E2 28322.628} C_VEL
LIN {X 0,Y 600.787,Z 785.715,A -85,B 0,C 180,E1 28321.952,E2 28321.952} C_VEL
LIN {X 0,Y 600.82,Z 765.974,A -85,B 0,C 180,E1 28321.49,E2 28321.49} C_VEL
LIN {X 0,Y 600.89,Z 737.655,A -85,B 0,C 180,E1 28321.058,E2 28321.058} C_VEL
LIN {X 0,Y 601.106,Z 503.572,A -85,B 0,C 180,E1 28317.889,E2 28317.889} C_VEL
LIN {X 0,Y 600.949,Z 455.297,A -85,B 0,C 180,E1 28317.207,E2 28317.207} C_VEL
LIN {X 0,Y 601.071,Z 404.863,A -85,B 0,C 180,E1 28314.227,E2 28314.227} C_VEL
LIN {X 0,Y 601.015,Z 394.113,A -85,B 0,C 180,E1 28313.569,E2 28313.569} C_VEL
LIN {X 0,Y 599.971,Z 391.167,A -85,B 0,C 180,E1 28313.257,E2 28313.257} C_VEL
LIN {X 0,Y 599.973,Z 391.001,A -85,B 0,C 180,E1 28310.093,E2 28310.093} C_VEL
LIN {X 0,Y 599.941,Z 390.998,A -85,B 0,C 180,E1 28307.023,E2 28307.023} C_VEL
LIN {X 0,Y 599.967,Z 391.002,A -85,B 0,C 180,E1 28303.757,E2 28303.757} C_VEL
LIN {X 0,Y 599.958,Z 390.996,A -85,B 0,C 180,E1 28300.538,E2 28300.538} C_VEL
LIN {X 0,Y 599.935,Z 391.002,A -85,B 0,C 180,E1 28297.347,E2 28297.347} C_VEL
LIN {X 0,Y 599.962,Z 390.997,A -85,B 0,C 180,E1 28294.255,E2 28294.255} C_VEL
LIN {X 0,Y 599.918,Z 391.002,A -85,B 0,C 180,E1 28291.063,E2 28291.063} C_VEL
LIN {X 0,Y 599.964,Z 390.999,A -85,B 0,C 180,E1 28288.032,E2 28288.032} C_VEL
LIN {X 0,Y 599.908,Z 391.003,A -85,B 0,C 180,E1 28284.94,E2 28284.94} C_VEL
LIN {X 0,Y 599.929,Z 391.002,A -85,B 0,C 180,E1 28282.092,E2 28282.092} C_VEL
LIN {X 0,Y 599.901,Z 391.003,A -85,B 0,C 180,E1 28278.865,E2 28278.865} C_VEL
LIN {X 0,Y 599.908,Z 391.004,A -85,B 0,C 180,E1 28276.061,E2 28276.061} C_VEL
LIN {X 0,Y 599.9,Z 391.004,A -85,B 0,C 180,E1 28272.807,E2 28272.807} C_VEL
LIN {X 0,Y 599.901,Z 391.004,A -85,B 0,C 180,E1 28270.079,E2 28270.079} C_VEL
LIN {X 0,Y 599.922,Z 391.002,A -85,B 0,C 180,E1 28266.796,E2 28266.796} C_VEL
LIN {X 0,Y 599.913,Z 391.003,A -85,B 0,C 180,E1 28263.918,E2 28263.918} C_VEL
LIN {X 0,Y 599.934,Z 391,A -85,B 0,C 180,E1 28260.668,E2 28260.668} C_VEL
LIN {X 0,Y 599.922,Z 391.002,A -85,B 0,C 180,E1 28257.803,E2 28257.803} C_VEL
LIN {X 0,Y 599.946,Z 390.998,A -85,B 0,C 180,E1 28254.549,E2 28254.549} C_VEL
LIN {X 0,Y 599.956,Z 391.003,A -85,B 0,C 180,E1 28253.391,E2 28253.391} C_VEL
LIN {X 0,Y 599.018,Z 391.128,A -85,B 0,C 180,E1 28252.656,E2 28252.656} C_VEL
LIN {X 0,Y 592.538,Z 391.923,A -85,B 0,C 180,E1 28250.592,E2 28250.592} C_VEL
LIN {X 0,Y 591.989,Z 391.988,A -85,B 0,C 180,E1 28250.054,E2 28250.054} C_VEL
LIN {X 0,Y 592.036,Z 391.99,A -85,B 0,C 180,E1 28246.92,E2 28246.92} C_VEL
LIN {X 0,Y 591.997,Z 391.988,A -85,B 0,C 180,E1 28243.818,E2 28243.818} C_VEL
LIN {X 0,Y 592.032,Z 391.988,A -85,B 0,C 180,E1 28240.669,E2 28240.669} C_VEL
LIN {X 0,Y 592.006,Z 391.987,A -85,B 0,C 180,E1 28237.485,E2 28237.485} C_VEL
LIN {X 0,Y 592.033,Z 391.986,A -85,B 0,C 180,E1 28234.276,E2 28234.276} C_VEL
LIN {X 0,Y 592.033,Z 391.989,A -85,B 0,C 180,E1 28231.007,E2 28231.007} C_VEL
LIN {X 0,Y 592.071,Z 392.261,A -85,B 0,C 180,E1 28229.866,E2 28229.866} C_VEL
LIN {X 0,Y 593.596,Z 396.939,A -85,B 0,C 180,E1 28229.392,E2 28229.392} C_VEL
LIN {X 0,Y 593.304,Z 439.834,A -85,B 0,C 180,E1 28226.269,E2 28226.269} C_VEL
LIN {X 0,Y 593.311,Z 452.82,A -85,B 0,C 180,E1 28225.372,E2 28225.372} C_VEL
LIN {X 0,Y 593.75,Z 457.222,A -85,B 0,C 180,E1 28225.286,E2 28225.286} C_VEL
LIN {X 0,Y 593.336,Z 713.948,A -85,B 0,C 180,E1 28221.875,E2 28221.875} C_VEL
LIN {X 0,Y 593.23,Z 734.232,A -85,B 0,C 180,E1 28221.422,E2 28221.422} C_VEL
LIN {X 0,Y 593.108,Z 753.468,A -85,B 0,C 180,E1 28220.823,E2 28220.823} C_VEL
LIN {X 0,Y 592.955,Z 773.256,A -85,B 0,C 180,E1 28220.025,E2 28220.025} C_VEL
LIN {X 0,Y 592.813,Z 792.118,A -85,B 0,C 180,E1 28219.074,E2 28219.074} C_VEL
LIN {X 0,Y 592.658,Z 810.853,A -85,B 0,C 180,E1 28217.924,E2 28217.924} C_VEL
LIN {X 0,Y 592.495,Z 828.525,A -85,B 0,C 180,E1 28216.62,E2 28216.62} C_VEL
LIN {X 0,Y 592.345,Z 844.501,A -85,B 0,C 180,E1 28215.226,E2 28215.226} C_VEL
LIN {X 0,Y 592.223,Z 859.142,A -85,B 0,C 180,E1 28213.73,E2 28213.73} C_VEL
LIN {X 0,Y 592.117,Z 872.817,A -85,B 0,C 180,E1 28212.092,E2 28212.092} C_VEL
LIN {X 0,Y 592.029,Z 885.454,A -85,B 0,C 180,E1 28210.299,E2 28210.299} C_VEL
LIN {X 0,Y 591.975,Z 896.44,A -85,B 0,C 180,E1 28208.426,E2 28208.426} C_VEL
LIN {X 0,Y 591.942,Z 905.271,A -85,B 0,C 180,E1 28206.598,E2 28206.598} C_VEL
LIN {X 0,Y 591.932,Z 912.782,A -85,B 0,C 180,E1 28204.652,E2 28204.652} C_VEL
LIN {X 0,Y 591.921,Z 918.393,A -85,B 0,C 180,E1 28202.716,E2 28202.716} C_VEL
LIN {X 0,Y 591.917,Z 922.344,A -85,B 0,C 180,E1 28200.782,E2 28200.782} C_VEL
LIN {X 0,Y 591.912,Z 924.768,A -85,B 0,C 180,E1 28198.753,E2 28198.753} C_VEL
LIN {X 0,Y 591.911,Z 925.472,A -85,B 0,C 180,E1 28196.806,E2 28196.806} C_VEL
LIN {X 0,Y 591.914,Z 924.487,A -85,B 0,C 180,E1 28194.763,E2 28194.763} C_VEL
LIN {X 0,Y 591.916,Z 921.704,A -85,B 0,C 180,E1 28192.735,E2 28192.735} C_VEL
LIN {X 0,Y 591.921,Z 917.301,A -85,B 0,C 180,E1 28190.774,E2 28190.774} C_VEL
LIN {X 0,Y 591.928,Z 911.196,A -85,B 0,C 180,E1 28188.819,E2 28188.819} C_VEL
LIN {X 0,Y 591.942,Z 903.844,A -85,B 0,C 180,E1 28186.988,E2 28186.988} C_VEL
LIN {X 0,Y 591.982,Z 894.813,A -85,B 0,C 180,E1 28185.174,E2 28185.174} C_VEL
LIN {X 0,Y 592.038,Z 883.938,A -85,B 0,C 180,E1 28183.375,E2 28183.375} C_VEL
LIN {X 0,Y 592.124,Z 871.532,A -85,B 0,C 180,E1 28181.652,E2 28181.652} C_VEL
LIN {X 0,Y 592.229,Z 857.6,A -85,B 0,C 180,E1 28180.012,E2 28180.012} C_VEL
LIN {X 0,Y 592.36,Z 841.879,A -85,B 0,C 180,E1 28178.442,E2 28178.442} C_VEL
LIN {X 0,Y 592.51,Z 825.113,A -85,B 0,C 180,E1 28177.025,E2 28177.025} C_VEL
LIN {X 0,Y 592.678,Z 807.339,A -85,B 0,C 180,E1 28175.759,E2 28175.759} C_VEL
LIN {X 0,Y 592.843,Z 789.444,A -85,B 0,C 180,E1 28174.69,E2 28174.69} C_VEL
LIN {X 0,Y 592.993,Z 770.706,A -85,B 0,C 180,E1 28173.768,E2 28173.768} C_VEL
LIN {X 0,Y 593.118,Z 751.536,A -85,B 0,C 180,E1 28173.018,E2 28173.018} C_VEL
LIN {X 0,Y 593.24,Z 731.286,A -85,B 0,C 180,E1 28172.413,E2 28172.413} C_VEL
LIN {X 0,Y 593.339,Z 710.639,A -85,B 0,C 180,E1 28171.984,E2 28171.984} C_VEL
LIN {X 0,Y 593.754,Z 455.134,A -85,B 0,C 180,E1 28168.596,E2 28168.596} C_VEL
LIN {X 0,Y 593.222,Z 451.962,A -85,B 0,C 180,E1 28168.501,E2 28168.501} C_VEL
LIN {X 0,Y 593.518,Z 408.368,A -85,B 0,C 180,E1 28165.36,E2 28165.36} C_VEL
LIN {X 0,Y 593.506,Z 396.604,A -85,B 0,C 180,E1 28164.488,E2 28164.488} C_VEL
LIN {X 0,Y 592.046,Z 392.165,A -85,B 0,C 180,E1 28164.024,E2 28164.024} C_VEL
LIN {X 0,Y 592.031,Z 391.985,A -85,B 0,C 180,E1 28160.766,E2 28160.766} C_VEL
LIN {X 0,Y 592.033,Z 391.982,A -85,B 0,C 180,E1 28157.465,E2 28157.465} C_VEL
LIN {X 0,Y 592.011,Z 391.988,A -85,B 0,C 180,E1 28154.22,E2 28154.22} C_VEL
LIN {X 0,Y 592.027,Z 391.984,A -85,B 0,C 180,E1 28151.045,E2 28151.045} C_VEL
LIN {X 0,Y 592.01,Z 391.982,A -85,B 0,C 180,E1 28147.873,E2 28147.873} C_VEL
LIN {X 0,Y 592.024,Z 391.987,A -85,B 0,C 180,E1 28144.703,E2 28144.703} C_VEL
LIN {X 0,Y 592.013,Z 391.987,A -85,B 0,C 180,E1 28141.556,E2 28141.556} C_VEL
LIN {X 0,Y 592.027,Z 391.988,A -85,B 0,C 180,E1 28138.314,E2 28138.314} C_VEL
LIN {X 0,Y 592.022,Z 391.982,A -85,B 0,C 180,E1 28135.072,E2 28135.072} C_VEL
LIN {X 0,Y 592.03,Z 391.99,A -85,B 0,C 180,E1 28131.696,E2 28131.696} C_VEL
LIN {X 0,Y 592.028,Z 391.984,A -85,B 0,C 180,E1 28128.414,E2 28128.414} C_VEL
LIN {X 0,Y 592.016,Z 391.988,A -85,B 0,C 180,E1 28125.182,E2 28125.182} C_VEL
LIN {X 0,Y 592.021,Z 391.985,A -85,B 0,C 180,E1 28121.975,E2 28121.975} C_VEL
LIN {X 0,Y 592.015,Z 391.986,A -85,B 0,C 180,E1 28118.799,E2 28118.799} C_VEL
LIN {X 0,Y 592.021,Z 391.986,A -85,B 0,C 180,E1 28115.639,E2 28115.639} C_VEL
LIN {X 0,Y 592.018,Z 391.984,A -85,B 0,C 180,E1 28112.485,E2 28112.485} C_VEL
LIN {X 0,Y 592.027,Z 391.989,A -85,B 0,C 180,E1 28109.215,E2 28109.215} C_VEL
LIN {X 0,Y 592.031,Z 391.98,A -85,B 0,C 180,E1 28105.939,E2 28105.939} C_VEL
LIN {X 0,Y 592.031,Z 391.991,A -85,B 0,C 180,E1 28102.648,E2 28102.648} C_VEL
LIN {X 0,Y 592.026,Z 391.981,A -85,B 0,C 180,E1 28099.434,E2 28099.434} C_VEL
LIN {X 0,Y 592.019,Z 391.987,A -85,B 0,C 180,E1 28096.181,E2 28096.181} C_VEL
LIN {X 0,Y 592.018,Z 391.985,A -85,B 0,C 180,E1 28092.967,E2 28092.967} C_VEL
LIN {X 0,Y 592.019,Z 391.985,A -85,B 0,C 180,E1 28089.822,E2 28089.822} C_VEL
LIN {X 0,Y 592.018,Z 391.987,A -85,B 0,C 180,E1 28086.595,E2 28086.595} C_VEL
LIN {X 0,Y 592.024,Z 391.982,A -85,B 0,C 180,E1 28083.389,E2 28083.389} C_VEL
LIN {X 0,Y 592.03,Z 391.991,A -85,B 0,C 180,E1 28080.097,E2 28080.097} C_VEL
LIN {X 0,Y 592.027,Z 391.982,A -85,B 0,C 180,E1 28076.708,E2 28076.708} C_VEL
LIN {X 0,Y 592.027,Z 391.988,A -85,B 0,C 180,E1 28073.503,E2 28073.503} C_VEL
LIN {X 0,Y 592.015,Z 391.985,A -85,B 0,C 180,E1 28070.277,E2 28070.277} C_VEL
LIN {X 0,Y 592.023,Z 391.988,A -85,B 0,C 180,E1 28067.119,E2 28067.119} C_VEL
LIN {X 0,Y 592.013,Z 391.986,A -85,B 0,C 180,E1 28063.92,E2 28063.92} C_VEL
LIN {X 0,Y 592.023,Z 391.986,A -85,B 0,C 180,E1 28060.75,E2 28060.75} C_VEL
LIN {X 0,Y 592.014,Z 391.988,A -85,B 0,C 180,E1 28057.562,E2 28057.562} C_VEL
LIN {X 0,Y 592.028,Z 391.984,A -85,B 0,C 180,E1 28054.383,E2 28054.383} C_VEL
LIN {X 0,Y 592.024,Z 391.99,A -85,B 0,C 180,E1 28051.117,E2 28051.117} C_VEL
LIN {X 0,Y 592.025,Z 391.982,A -85,B 0,C 180,E1 28047.746,E2 28047.746} C_VEL
LIN {X 0,Y 592.03,Z 391.991,A -85,B 0,C 180,E1 28044.482,E2 28044.482} C_VEL
LIN {X 0,Y 592.013,Z 391.985,A -85,B 0,C 180,E1 28041.287,E2 28041.287} C_VEL
LIN {X 0,Y 592.026,Z 391.989,A -85,B 0,C 180,E1 28038.142,E2 28038.142} C_VEL
LIN {X 0,Y 592.01,Z 391.984,A -85,B 0,C 180,E1 28034.956,E2 28034.956} C_VEL
LIN {X 0,Y 592.024,Z 391.983,A -85,B 0,C 180,E1 28031.845,E2 28031.845} C_VEL
LIN {X 0,Y 592.008,Z 391.985,A -85,B 0,C 180,E1 28028.676,E2 28028.676} C_VEL
LIN {X 0,Y 592.069,Z 392.233,A -85,B 0,C 180,E1 28027.237,E2 28027.237} C_VEL
LIN {X 0,Y 593.963,Z 397.122,A -85,B 0,C 180,E1 28026.748,E2 28026.748} C_VEL
LIN {X 0,Y 594.304,Z 399.223,A -85,B 0,C 180,E1 28026.593,E2 28026.593} C_VEL
LIN {X 0,Y 593.935,Z 450.199,A -85,B 0,C 180,E1 28023.517,E2 28023.517} C_VEL
LIN {X 0,Y 594.061,Z 455.926,A -85,B 0,C 180,E1 28023.21,E2 28023.21} C_VEL
LIN {X 0,Y 594.398,Z 460.908,A -85,B 0,C 180,E1 28023.119,E2 28023.119} C_VEL
LIN {X 0,Y 593.983,Z 681.166,A -85,B 0,C 180,E1 28020.081,E2 28020.081} C_VEL
LIN {X 0,Y 593.809,Z 761.751,A -85,B 0,C 180,E1 28018.963,E2 28018.963} C_VEL
LIN {X 0,Y 593.688,Z 782.68,A -85,B 0,C 180,E1 28018.493,E2 28018.493} C_VEL
LIN {X 0,Y 593.537,Z 803.389,A -85,B 0,C 180,E1 28017.866,E2 28017.866} C_VEL
LIN {X 0,Y 593.382,Z 823.817,A -85,B 0,C 180,E1 28017.063,E2 28017.063} C_VEL
LIN {X 0,Y 593.182,Z 843.721,A -85,B 0,C 180,E1 28016.101,E2 28016.101} C_VEL
LIN {X 0,Y 593.005,Z 863.081,A -85,B 0,C 180,E1 28014.985,E2 28014.985} C_VEL
LIN {X 0,Y 592.806,Z 881.616,A -85,B 0,C 180,E1 28013.716,E2 28013.716} C_VEL
LIN {X 0,Y 592.599,Z 899.859,A -85,B 0,C 180,E1 28012.26,E2 28012.26} C_VEL
LIN {X 0,Y 592.419,Z 917.141,A -85,B 0,C 180,E1 28010.657,E2 28010.657} C_VEL
LIN {X 0,Y 592.298,Z 932.453,A -85,B 0,C 180,E1 28009.016,E2 28009.016} C_VEL
LIN {X 0,Y 592.173,Z 947.099,A -85,B 0,C 180,E1 28007.188,E2 28007.188} C_VEL
LIN {X 0,Y 592.071,Z 959.626,A -85,B 0,C 180,E1 28005.362,E2 28005.362} C_VEL
LIN {X 0,Y 592,Z 971.242,A -85,B 0,C 180,E1 28003.38,E2 28003.38} C_VEL
LIN {X 0,Y 591.953,Z 980.516,A -85,B 0,C 180,E1 28001.498,E2 28001.498} C_VEL
LIN {X 0,Y 591.917,Z 988.458,A -85,B 0,C 180,E1 27999.53,E2 27999.53} C_VEL
LIN {X 0,Y 591.909,Z 994.867,A -85,B 0,C 180,E1 27997.573,E2 27997.573} C_VEL
LIN {X 0,Y 591.911,Z 999.805,A -85,B 0,C 180,E1 27995.527,E2 27995.527} C_VEL
LIN {X 0,Y 591.915,Z 1003.4,A -85,B 0,C 180,E1 27993.333,E2 27993.333} C_VEL
LIN {X 0,Y 591.908,Z 1005.209,A -85,B 0,C 180,E1 27991.26,E2 27991.26} C_VEL
LIN {X 0,Y 591.894,Z 1005.329,A -85,B 0,C 180,E1 27989.228,E2 27989.228} C_VEL
LIN {X 0,Y 591.892,Z 1003.898,A -85,B 0,C 180,E1 27987.097,E2 27987.097} C_VEL
LIN {X 0,Y 591.896,Z 1001.149,A -85,B 0,C 180,E1 27985.157,E2 27985.157} C_VEL
LIN {X 0,Y 591.914,Z 996.658,A -85,B 0,C 180,E1 27983.114,E2 27983.114} C_VEL
LIN {X 0,Y 591.936,Z 990.6,A -85,B 0,C 180,E1 27981.062,E2 27981.062} C_VEL
LIN {X 0,Y 591.95,Z 983.075,A -85,B 0,C 180,E1 27979.098,E2 27979.098} C_VEL
LIN {X 0,Y 591.994,Z 973.341,A -85,B 0,C 180,E1 27977.021,E2 27977.021} C_VEL
LIN {X 0,Y 592.064,Z 962.759,A -85,B 0,C 180,E1 27975.129,E2 27975.129} C_VEL
LIN {X 0,Y 592.146,Z 950.055,A -85,B 0,C 180,E1 27973.22,E2 27973.22} C_VEL
LIN {X 0,Y 592.256,Z 935.89,A -85,B 0,C 180,E1 27971.396,E2 27971.396} C_VEL
LIN {X 0,Y 592.406,Z 920.222,A -85,B 0,C 180,E1 27969.657,E2 27969.657} C_VEL
LIN {X 0,Y 592.578,Z 904.135,A -85,B 0,C 180,E1 27968.109,E2 27968.109} C_VEL
LIN {X 0,Y 592.743,Z 886.5,A -85,B 0,C 180,E1 27966.649,E2 27966.649} C_VEL
LIN {X 0,Y 592.937,Z 868.261,A -85,B 0,C 180,E1 27965.354,E2 27965.354} C_VEL
LIN {X 0,Y 593.156,Z 848.879,A -85,B 0,C 180,E1 27964.176,E2 27964.176} C_VEL
LIN {X 0,Y 593.295,Z 829.867,A -85,B 0,C 180,E1 27963.208,E2 27963.208} C_VEL
LIN {X 0,Y 593.507,Z 808.591,A -85,B 0,C 180,E1 27962.325,E2 27962.325} C_VEL
LIN {X 0,Y 593.681,Z 787.794,A -85,B 0,C 180,E1 27961.641,E2 27961.641} C_VEL
LIN {X 0,Y 593.764,Z 767.207,A -85,B 0,C 180,E1 27961.146,E2 27961.146} C_VEL
LIN {X 0,Y 593.882,Z 739.757,A -85,B 0,C 180,E1 27960.712,E2 27960.712} C_VEL
LIN {X 0,Y 594.322,Z 506.321,A -85,B 0,C 180,E1 27957.516,E2 27957.516} C_VEL
LIN {X 0,Y 594.207,Z 456.747,A -85,B 0,C 180,E1 27956.81,E2 27956.81} C_VEL
LIN {X 0,Y 593.913,Z 454.156,A -85,B 0,C 180,E1 27956.717,E2 27956.717} C_VEL
LIN {X 0,Y 594.278,Z 402.829,A -85,B 0,C 180,E1 27953.629,E2 27953.629} C_VEL
LIN {X 0,Y 594.311,Z 397.987,A -85,B 0,C 180,E1 27953.331,E2 27953.331} C_VEL
LIN {X 0,Y 592.076,Z 392.278,A -85,B 0,C 180,E1 27952.776,E2 27952.776} C_VEL
LIN {X 0,Y 592.025,Z 391.968,A -85,B 0,C 180,E1 27951.824,E2 27951.824} C_VEL
LIN {X 0,Y 592.039,Z 391.983,A -85,B 0,C 180,E1 27948.55,E2 27948.55} C_VEL
LIN {X 0,Y 591.999,Z 391.99,A -85,B 0,C 180,E1 27945.32,E2 27945.32} C_VEL
LIN {X 0,Y 592.035,Z 391.985,A -85,B 0,C 180,E1 27942.154,E2 27942.154} C_VEL
LIN {X 0,Y 591.989,Z 391.989,A -85,B 0,C 180,E1 27939.025,E2 27939.025} C_VEL
LIN {X 0,Y 592.038,Z 391.991,A -85,B 0,C 180,E1 27935.847,E2 27935.847} C_VEL
LIN {X 0,Y 591.981,Z 391.989,A -85,B 0,C 180,E1 27932.748,E2 27932.748} C_VEL
LIN {X 0,Y 592.023,Z 391.993,A -85,B 0,C 180,E1 27929.548,E2 27929.548} C_VEL
LIN {X 0,Y 591.97,Z 391.989,A -85,B 0,C 180,E1 27926.589,E2 27926.589} C_VEL
LIN {X 0,Y 592.023,Z 391.993,A -85,B 0,C 180,E1 27923.489,E2 27923.489} C_VEL
LIN {X 0,Y 591.96,Z 391.991,A -85,B 0,C 180,E1 27920.465,E2 27920.465} C_VEL
LIN {X 0,Y 592.004,Z 391.993,A -85,B 0,C 180,E1 27917.292,E2 27917.292} C_VEL
LIN {X 0,Y 591.949,Z 391.992,A -85,B 0,C 180,E1 27914.376,E2 27914.376} C_VEL
LIN {X 0,Y 592.026,Z 391.992,A -85,B 0,C 180,E1 27911.298,E2 27911.298} C_VEL
LIN {X 0,Y 591.958,Z 391.991,A -85,B 0,C 180,E1 27908.254,E2 27908.254} C_VEL
LIN {X 0,Y 592.029,Z 391.99,A -85,B 0,C 180,E1 27905.135,E2 27905.135} C_VEL
LIN {X 0,Y 591.968,Z 391.99,A -85,B 0,C 180,E1 27902.129,E2 27902.129} C_VEL
LIN {X 0,Y 592.037,Z 391.989,A -85,B 0,C 180,E1 27899.032,E2 27899.032} C_VEL
LIN {X 0,Y 591.98,Z 391.989,A -85,B 0,C 180,E1 27895.932,E2 27895.932} C_VEL
LIN {X 0,Y 592.033,Z 391.986,A -85,B 0,C 180,E1 27892.723,E2 27892.723} C_VEL
LIN {X 0,Y 591.989,Z 391.988,A -85,B 0,C 180,E1 27890.054,E2 27890.054} C_VEL
LIN {X 0,Y 591,Z 392.121,A -85,B 0,C 180,E1 27889.309,E2 27889.309} C_VEL
LIN {X 0,Y 584.622,Z 392.916,A -85,B 0,C 180,E1 27887.216,E2 27887.216} C_VEL
LIN {X 0,Y 584.099,Z 392.975,A -85,B 0,C 180,E1 27886.672,E2 27886.672} C_VEL
LIN {X 0,Y 584.067,Z 392.98,A -85,B 0,C 180,E1 27883.454,E2 27883.454} C_VEL
LIN {X 0,Y 584.078,Z 392.975,A -85,B 0,C 180,E1 27880.083,E2 27880.083} C_VEL
LIN {X 0,Y 584.094,Z 392.98,A -85,B 0,C 180,E1 27876.806,E2 27876.806} C_VEL
LIN {X 0,Y 584.072,Z 392.979,A -85,B 0,C 180,E1 27873.54,E2 27873.54} C_VEL
LIN {X 0,Y 584.099,Z 393.073,A -85,B 0,C 180,E1 27870.349,E2 27870.349} C_VEL
LIN {X 0,Y 584.461,Z 394.564,A -85,B 0,C 180,E1 27870.144,E2 27870.144} C_VEL
LIN {X 0,Y 586.446,Z 400.372,A -85,B 0,C 180,E1 27869.577,E2 27869.577} C_VEL
LIN {X 0,Y 586.004,Z 443.003,A -85,B 0,C 180,E1 27866.439,E2 27866.439} C_VEL
LIN {X 0,Y 585.992,Z 452.79,A -85,B 0,C 180,E1 27865.761,E2 27865.761} C_VEL
LIN {X 0,Y 586.704,Z 457.972,A -85,B 0,C 180,E1 27865.648,E2 27865.648} C_VEL
LIN {X 0,Y 586.076,Z 713.877,A -85,B 0,C 180,E1 27862.206,E2 27862.206} C_VEL
LIN {X 0,Y 585.919,Z 734.284,A -85,B 0,C 180,E1 27861.747,E2 27861.747} C_VEL
LIN {X 0,Y 585.731,Z 753.388,A -85,B 0,C 180,E1 27861.146,E2 27861.146} C_VEL
LIN {X 0,Y 585.518,Z 772.69,A -85,B 0,C 180,E1 27860.362,E2 27860.362} C_VEL
LIN {X 0,Y 585.299,Z 791.768,A -85,B 0,C 180,E1 27859.393,E2 27859.393} C_VEL
LIN {X 0,Y 585.059,Z 809.892,A -85,B 0,C 180,E1 27858.274,E2 27858.274} C_VEL
LIN {X 0,Y 584.807,Z 827.312,A -85,B 0,C 180,E1 27856.985,E2 27856.985} C_VEL
LIN {X 0,Y 584.586,Z 843.457,A -85,B 0,C 180,E1 27855.575,E2 27855.575} C_VEL
LIN {X 0,Y 584.388,Z 858.249,A -85,B 0,C 180,E1 27854.061,E2 27854.061} C_VEL
LIN {X 0,Y 584.231,Z 872.104,A -85,B 0,C 180,E1 27852.395,E2 27852.395} C_VEL
LIN {X 0,Y 584.117,Z 884.178,A -85,B 0,C 180,E1 27850.685,E2 27850.685} C_VEL
LIN {X 0,Y 584.032,Z 894.701,A -85,B 0,C 180,E1 27848.921,E2 27848.921} C_VEL
LIN {X 0,Y 583.97,Z 903.848,A -85,B 0,C 180,E1 27847.058,E2 27847.058} C_VEL
LIN {X 0,Y 583.943,Z 911.071,A -85,B 0,C 180,E1 27845.238,E2 27845.238} C_VEL
LIN {X 0,Y 583.924,Z 917.299,A -85,B 0,C 180,E1 27843.222,E2 27843.222} C_VEL
LIN {X 0,Y 583.912,Z 921.674,A -85,B 0,C 180,E1 27841.251,E2 27841.251} C_VEL
LIN {X 0,Y 583.909,Z 924.506,A -85,B 0,C 180,E1 27839.155,E2 27839.155} C_VEL
LIN {X 0,Y 583.91,Z 925.479,A -85,B 0,C 180,E1 27837.073,E2 27837.073} C_VEL
LIN {X 0,Y 583.913,Z 924.722,A -85,B 0,C 180,E1 27835.064,E2 27835.064} C_VEL
LIN {X 0,Y 583.918,Z 922.357,A -85,B 0,C 180,E1 27833.084,E2 27833.084} C_VEL
LIN {X 0,Y 583.924,Z 918.25,A -85,B 0,C 180,E1 27831.058,E2 27831.058} C_VEL
LIN {X 0,Y 583.936,Z 912.552,A -85,B 0,C 180,E1 27829.087,E2 27829.087} C_VEL
LIN {X 0,Y 583.96,Z 905.051,A -85,B 0,C 180,E1 27827.125,E2 27827.125} C_VEL
LIN {X 0,Y 584.009,Z 896.23,A -85,B 0,C 180,E1 27825.285,E2 27825.285} C_VEL
LIN {X 0,Y 584.094,Z 885.668,A -85,B 0,C 180,E1 27823.46,E2 27823.46} C_VEL
LIN {X 0,Y 584.227,Z 873.121,A -85,B 0,C 180,E1 27821.648,E2 27821.648} C_VEL
LIN {X 0,Y 584.383,Z 860.048,A -85,B 0,C 180,E1 27820.048,E2 27820.048} C_VEL
LIN {X 0,Y 584.57,Z 845.295,A -85,B 0,C 180,E1 27818.506,E2 27818.506} C_VEL
LIN {X 0,Y 584.8,Z 828.519,A -85,B 0,C 180,E1 27817.019,E2 27817.019} C_VEL
LIN {X 0,Y 585.052,Z 810.647,A -85,B 0,C 180,E1 27815.686,E2 27815.686} C_VEL
LIN {X 0,Y 585.286,Z 792.41,A -85,B 0,C 180,E1 27814.554,E2 27814.554} C_VEL
LIN {X 0,Y 585.493,Z 774.241,A -85,B 0,C 180,E1 27813.62,E2 27813.62} C_VEL
LIN {X 0,Y 585.732,Z 754.003,A -85,B 0,C 180,E1 27812.786,E2 27812.786} C_VEL
LIN {X 0,Y 585.921,Z 733.869,A -85,B 0,C 180,E1 27812.152,E2 27812.152} C_VEL
LIN {X 0,Y 586.076,Z 713.624,A -85,B 0,C 180,E1 27811.7,E2 27811.7} C_VEL
LIN {X 0,Y 586.707,Z 457.453,A -85,B 0,C 180,E1 27808.255,E2 27808.255} C_VEL
LIN {X 0,Y 585.911,Z 452.007,A -85,B 0,C 180,E1 27808.115,E2 27808.115} C_VEL
LIN {X 0,Y 586.349,Z 409.448,A -85,B 0,C 180,E1 27805.009,E2 27805.009} C_VEL
LIN {X 0,Y 586.369,Z 399.649,A -85,B 0,C 180,E1 27804.273,E2 27804.273} C_VEL
LIN {X 0,Y 584.121,Z 393.17,A -85,B 0,C 180,E1 27803.598,E2 27803.598} C_VEL
LIN {X 0,Y 584.071,Z 392.977,A -85,B 0,C 180,E1 27800.34,E2 27800.34} C_VEL
LIN {X 0,Y 584.087,Z 392.972,A -85,B 0,C 180,E1 27797.14,E2 27797.14} C_VEL
LIN {X 0,Y 584.07,Z 392.974,A -85,B 0,C 180,E1 27794,E2 27794} C_VEL
LIN {X 0,Y 584.088,Z 392.975,A -85,B 0,C 180,E1 27790.81,E2 27790.81} C_VEL
LIN {X 0,Y 584.078,Z 392.966,A -85,B 0,C 180,E1 27787.557,E2 27787.557} C_VEL
LIN {X 0,Y 584.094,Z 392.982,A -85,B 0,C 180,E1 27784.213,E2 27784.213} C_VEL
LIN {X 0,Y 584.093,Z 392.972,A -85,B 0,C 180,E1 27780.91,E2 27780.91} C_VEL
LIN {X 0,Y 584.076,Z 392.978,A -85,B 0,C 180,E1 27777.6,E2 27777.6} C_VEL
LIN {X 0,Y 584.085,Z 392.973,A -85,B 0,C 180,E1 27774.403,E2 27774.403} C_VEL
LIN {X 0,Y 584.076,Z 392.972,A -85,B 0,C 180,E1 27771.16,E2 27771.16} C_VEL
LIN {X 0,Y 584.086,Z 392.978,A -85,B 0,C 180,E1 27767.983,E2 27767.983} C_VEL
LIN {X 0,Y 584.085,Z 392.972,A -85,B 0,C 180,E1 27764.714,E2 27764.714} C_VEL
LIN {X 0,Y 584.094,Z 392.98,A -85,B 0,C 180,E1 27761.358,E2 27761.358} C_VEL
LIN {X 0,Y 584.088,Z 392.972,A -85,B 0,C 180,E1 27758.044,E2 27758.044} C_VEL
LIN {X 0,Y 584.077,Z 392.977,A -85,B 0,C 180,E1 27754.754,E2 27754.754} C_VEL
LIN {X 0,Y 584.081,Z 392.974,A -85,B 0,C 180,E1 27751.59,E2 27751.59} C_VEL
LIN {X 0,Y 584.077,Z 392.975,A -85,B 0,C 180,E1 27748.418,E2 27748.418} C_VEL
LIN {X 0,Y 584.082,Z 392.974,A -85,B 0,C 180,E1 27745.23,E2 27745.23} C_VEL
LIN {X 0,Y 584.084,Z 392.972,A -85,B 0,C 180,E1 27742.018,E2 27742.018} C_VEL
LIN {X 0,Y 584.096,Z 392.979,A -85,B 0,C 180,E1 27738.67,E2 27738.67} C_VEL
LIN {X 0,Y 584.087,Z 392.971,A -85,B 0,C 180,E1 27735.285,E2 27735.285} C_VEL
LIN {X 0,Y 584.083,Z 392.978,A -85,B 0,C 180,E1 27732.055,E2 27732.055} C_VEL
LIN {X 0,Y 584.079,Z 392.972,A -85,B 0,C 180,E1 27728.863,E2 27728.863} C_VEL
LIN {X 0,Y 584.081,Z 392.976,A -85,B 0,C 180,E1 27725.698,E2 27725.698} C_VEL
LIN {X 0,Y 584.078,Z 392.974,A -85,B 0,C 180,E1 27722.453,E2 27722.453} C_VEL
LIN {X 0,Y 584.087,Z 392.971,A -85,B 0,C 180,E1 27719.216,E2 27719.216} C_VEL
LIN {X 0,Y 584.093,Z 392.98,A -85,B 0,C 180,E1 27715.877,E2 27715.877} C_VEL
LIN {X 0,Y 584.085,Z 392.969,A -85,B 0,C 180,E1 27712.525,E2 27712.525} C_VEL
LIN {X 0,Y 584.085,Z 392.976,A -85,B 0,C 180,E1 27709.246,E2 27709.246} C_VEL
LIN {X 0,Y 584.075,Z 392.975,A -85,B 0,C 180,E1 27706.033,E2 27706.033} C_VEL
LIN {X 0,Y 584.084,Z 392.975,A -85,B 0,C 180,E1 27702.877,E2 27702.877} C_VEL
LIN {X 0,Y 584.075,Z 392.977,A -85,B 0,C 180,E1 27699.665,E2 27699.665} C_VEL
LIN {X 0,Y 584.091,Z 392.972,A -85,B 0,C 180,E1 27696.387,E2 27696.387} C_VEL
LIN {X 0,Y 584.095,Z 392.982,A -85,B 0,C 180,E1 27693.024,E2 27693.024} C_VEL
LIN {X 0,Y 584.078,Z 392.974,A -85,B 0,C 180,E1 27689.669,E2 27689.669} C_VEL
LIN {X 0,Y 584.087,Z 392.978,A -85,B 0,C 180,E1 27686.433,E2 27686.433} C_VEL
LIN {X 0,Y 584.072,Z 392.976,A -85,B 0,C 180,E1 27683.242,E2 27683.242} C_VEL
LIN {X 0,Y 584.086,Z 392.974,A -85,B 0,C 180,E1 27680.064,E2 27680.064} C_VEL
LIN {X 0,Y 584.073,Z 392.978,A -85,B 0,C 180,E1 27676.825,E2 27676.825} C_VEL
LIN {X 0,Y 584.094,Z 392.974,A -85,B 0,C 180,E1 27673.607,E2 27673.607} C_VEL
LIN {X 0,Y 584.086,Z 392.979,A -85,B 0,C 180,E1 27670.322,E2 27670.322} C_VEL
LIN {X 0,Y 584.124,Z 393.207,A -85,B 0,C 180,E1 27667.772,E2 27667.772} C_VEL
LIN {X 0,Y 585.853,Z 397.535,A -85,B 0,C 180,E1 27667.316,E2 27667.316} C_VEL
LIN {X 0,Y 587.526,Z 401.778,A -85,B 0,C 180,E1 27666.924,E2 27666.924} C_VEL
LIN {X 0,Y 586.969,Z 452.811,A -85,B 0,C 180,E1 27663.81,E2 27663.81} C_VEL
LIN {X 0,Y 587.164,Z 456.23,A -85,B 0,C 180,E1 27663.648,E2 27663.648} C_VEL
LIN {X 0,Y 587.694,Z 461.097,A -85,B 0,C 180,E1 27663.543,E2 27663.543} C_VEL
LIN {X 0,Y 587.058,Z 681.672,A -85,B 0,C 180,E1 27660.467,E2 27660.467} C_VEL
LIN {X 0,Y 586.801,Z 761.858,A -85,B 0,C 180,E1 27659.341,E2 27659.341} C_VEL
LIN {X 0,Y 586.615,Z 782.94,A -85,B 0,C 180,E1 27658.862,E2 27658.862} C_VEL
LIN {X 0,Y 586.372,Z 804.718,A -85,B 0,C 180,E1 27658.187,E2 27658.187} C_VEL
LIN {X 0,Y 586.144,Z 825.093,A -85,B 0,C 180,E1 27657.37,E2 27657.37} C_VEL
LIN {X 0,Y 585.832,Z 845.456,A -85,B 0,C 180,E1 27656.359,E2 27656.359} C_VEL
LIN {X 0,Y 585.522,Z 865.508,A -85,B 0,C 180,E1 27655.165,E2 27655.165} C_VEL
LIN {X 0,Y 585.25,Z 884.434,A -85,B 0,C 180,E1 27653.833,E2 27653.833} C_VEL
LIN {X 0,Y 584.945,Z 902.094,A -85,B 0,C 180,E1 27652.371,E2 27652.371} C_VEL
LIN {X 0,Y 584.675,Z 918.659,A -85,B 0,C 180,E1 27650.786,E2 27650.786} C_VEL
LIN {X 0,Y 584.472,Z 934.154,A -85,B 0,C 180,E1 27649.073,E2 27649.073} C_VEL
LIN {X 0,Y 584.299,Z 948.612,A -85,B 0,C 180,E1 27647.221,E2 27647.221} C_VEL
LIN {X 0,Y 584.156,Z 961.46,A -85,B 0,C 180,E1 27645.285,E2 27645.285} C_VEL
LIN {X 0,Y 584.048,Z 972.281,A -85,B 0,C 180,E1 27643.364,E2 27643.364} C_VEL
LIN {X 0,Y 583.981,Z 981.836,A -85,B 0,C 180,E1 27641.357,E2 27641.357} C_VEL
LIN {X 0,Y 583.931,Z 989.523,A -85,B 0,C 180,E1 27639.364,E2 27639.364} C_VEL
LIN {X 0,Y 583.903,Z 995.885,A -85,B 0,C 180,E1 27637.282,E2 27637.282} C_VEL
LIN {X 0,Y 583.9,Z 1000.423,A -85,B 0,C 180,E1 27635.308,E2 27635.308} C_VEL
LIN {X 0,Y 583.909,Z 1003.557,A -85,B 0,C 180,E1 27633.241,E2 27633.241} C_VEL
LIN {X 0,Y 583.913,Z 1005.261,A -85,B 0,C 180,E1 27631.081,E2 27631.081} C_VEL
LIN {X 0,Y 583.905,Z 1005.285,A -85,B 0,C 180,E1 27629.021,E2 27629.021} C_VEL
LIN {X 0,Y 583.902,Z 1003.674,A -85,B 0,C 180,E1 27626.861,E2 27626.861} C_VEL
LIN {X 0,Y 583.896,Z 1000.636,A -85,B 0,C 180,E1 27624.795,E2 27624.795} C_VEL
LIN {X 0,Y 583.904,Z 996.15,A -85,B 0,C 180,E1 27622.821,E2 27622.821} C_VEL
LIN {X 0,Y 583.934,Z 989.892,A -85,B 0,C 180,E1 27620.74,E2 27620.74} C_VEL
LIN {X 0,Y 583.979,Z 982.597,A -85,B 0,C 180,E1 27618.83,E2 27618.83} C_VEL
LIN {X 0,Y 584.044,Z 973.342,A -85,B 0,C 180,E1 27616.841,E2 27616.841} C_VEL
LIN {X 0,Y 584.151,Z 962.465,A -85,B 0,C 180,E1 27614.876,E2 27614.876} C_VEL
LIN {X 0,Y 584.275,Z 950.056,A -85,B 0,C 180,E1 27612.987,E2 27612.987} C_VEL
LIN {X 0,Y 584.444,Z 935.89,A -85,B 0,C 180,E1 27611.138,E2 27611.138} C_VEL
LIN {X 0,Y 584.663,Z 920.221,A -85,B 0,C 180,E1 27609.375,E2 27609.375} C_VEL
LIN {X 0,Y 584.927,Z 904.137,A -85,B 0,C 180,E1 27607.807,E2 27607.807} C_VEL
LIN {X 0,Y 585.202,Z 886.343,A -85,B 0,C 180,E1 27606.318,E2 27606.318} C_VEL
LIN {X 0,Y 585.472,Z 868.302,A -85,B 0,C 180,E1 27605.021,E2 27605.021} C_VEL
LIN {X 0,Y 585.806,Z 848.781,A -85,B 0,C 180,E1 27603.822,E2 27603.822} C_VEL
LIN {X 0,Y 586.039,Z 829.868,A -85,B 0,C 180,E1 27602.849,E2 27602.849} C_VEL
LIN {X 0,Y 586.338,Z 808.52,A -85,B 0,C 180,E1 27601.954,E2 27601.954} C_VEL
LIN {X 0,Y 586.6,Z 787.535,A -85,B 0,C 180,E1 27601.26,E2 27601.26} C_VEL
LIN {X 0,Y 586.735,Z 766.883,A -85,B 0,C 180,E1 27600.76,E2 27600.76} C_VEL
LIN {X 0,Y 586.905,Z 738.981,A -85,B 0,C 180,E1 27600.319,E2 27600.319} C_VEL
LIN {X 0,Y 587.572,Z 505.176,A -85,B 0,C 180,E1 27597.08,E2 27597.08} C_VEL
LIN {X 0,Y 587.494,Z 458.116,A -85,B 0,C 180,E1 27596.401,E2 27596.401} C_VEL
LIN {X 0,Y 586.956,Z 454.156,A -85,B 0,C 180,E1 27596.27,E2 27596.27} C_VEL
LIN {X 0,Y 587.503,Z 403.798,A -85,B 0,C 180,E1 27593.201,E2 27593.201} C_VEL
LIN {X 0,Y 587.263,Z 400.68,A -85,B 0,C 180,E1 27592.987,E2 27592.987} C_VEL
LIN {X 0,Y 584.147,Z 393.339,A -85,B 0,C 180,E1 27592.259,E2 27592.259} C_VEL
LIN {X 0,Y 584.07,Z 392.954,A -85,B 0,C 180,E1 27591.585,E2 27591.585} C_VEL
LIN {X 0,Y 584.094,Z 392.972,A -85,B 0,C 180,E1 27588.385,E2 27588.385} C_VEL
LIN {X 0,Y 584.059,Z 392.979,A -85,B 0,C 180,E1 27585.271,E2 27585.271} C_VEL
LIN {X 0,Y 584.096,Z 392.973,A -85,B 0,C 180,E1 27582.146,E2 27582.146} C_VEL
LIN {X 0,Y 584.051,Z 392.978,A -85,B 0,C 180,E1 27578.999,E2 27578.999} C_VEL
LIN {X 0,Y 584.099,Z 392.981,A -85,B 0,C 180,E1 27575.774,E2 27575.774} C_VEL
LIN {X 0,Y 584.047,Z 392.978,A -85,B 0,C 180,E1 27572.625,E2 27572.625} C_VEL
LIN {X 0,Y 584.057,Z 392.981,A -85,B 0,C 180,E1 27569.315,E2 27569.315} C_VEL
LIN {X 0,Y 584.04,Z 392.978,A -85,B 0,C 180,E1 27566.43,E2 27566.43} C_VEL
LIN {X 0,Y 584.039,Z 392.982,A -85,B 0,C 180,E1 27563.081,E2 27563.081} C_VEL
LIN {X 0,Y 584.032,Z 392.98,A -85,B 0,C 180,E1 27560.232,E2 27560.232} C_VEL
LIN {X 0,Y 584.023,Z 392.982,A -85,B 0,C 180,E1 27556.873,E2 27556.873} C_VEL
LIN {X 0,Y 584.024,Z 392.981,A -85,B 0,C 180,E1 27554.07,E2 27554.07} C_VEL
LIN {X 0,Y 584.026,Z 392.981,A -85,B 0,C 180,E1 27550.755,E2 27550.755} C_VEL
LIN {X 0,Y 584.039,Z 392.98,A -85,B 0,C 180,E1 27547.872,E2 27547.872} C_VEL
LIN {X 0,Y 584.038,Z 392.979,A -85,B 0,C 180,E1 27544.615,E2 27544.615} C_VEL
LIN {X 0,Y 584.056,Z 392.98,A -85,B 0,C 180,E1 27541.667,E2 27541.667} C_VEL
LIN {X 0,Y 584.045,Z 392.978,A -85,B 0,C 180,E1 27538.43,E2 27538.43} C_VEL
LIN {X 0,Y 584.08,Z 392.98,A -85,B 0,C 180,E1 27535.385,E2 27535.385} C_VEL
LIN {X 0,Y 584.048,Z 392.978,A -85,B 0,C 180,E1 27532.128,E2 27532.128} C_VEL
LIN {X 0,Y 584.098,Z 392.979,A -85,B 0,C 180,E1 27528.946,E2 27528.946} C_VEL
LIN {X 0,Y 584.099,Z 392.975,A -85,B 0,C 180,E1 27526.672,E2 27526.672} C_VEL
LIN {X 0,Y 583.106,Z 393.097,A -85,B 0,C 180,E1 27525.916,E2 27525.916} C_VEL
LIN {X 0,Y 576.655,Z 393.902,A -85,B 0,C 180,E1 27523.796,E2 27523.796} C_VEL
LIN {X 0,Y 576.145,Z 393.97,A -85,B 0,C 180,E1 27523.244,E2 27523.244} C_VEL
LIN {X 0,Y 576.13,Z 393.966,A -85,B 0,C 180,E1 27519.902,E2 27519.902} C_VEL
LIN {X 0,Y 576.153,Z 393.968,A -85,B 0,C 180,E1 27516.692,E2 27516.692} C_VEL
LIN {X 0,Y 576.136,Z 393.971,A -85,B 0,C 180,E1 27513.4,E2 27513.4} C_VEL
LIN {X 0,Y 576.182,Z 394.17,A -85,B 0,C 180,E1 27510.764,E2 27510.764} C_VEL
LIN {X 0,Y 577.519,Z 398.12,A -85,B 0,C 180,E1 27510.32,E2 27510.32} C_VEL
LIN {X 0,Y 579.304,Z 403.471,A -85,B 0,C 180,E1 27509.793,E2 27509.793} C_VEL
LIN {X 0,Y 578.702,Z 446.264,A -85,B 0,C 180,E1 27506.607,E2 27506.607} C_VEL
LIN {X 0,Y 578.732,Z 452.948,A -85,B 0,C 180,E1 27506.154,E2 27506.154} C_VEL
LIN {X 0,Y 579.68,Z 459.267,A -85,B 0,C 180,E1 27506.01,E2 27506.01} C_VEL
LIN {X 0,Y 578.835,Z 713.786,A -85,B 0,C 180,E1 27502.546,E2 27502.546} C_VEL
LIN {X 0,Y 578.629,Z 734.191,A -85,B 0,C 180,E1 27502.083,E2 27502.083} C_VEL
LIN {X 0,Y 578.368,Z 754.092,A -85,B 0,C 180,E1 27501.448,E2 27501.448} C_VEL
LIN {X 0,Y 578.074,Z 773.725,A -85,B 0,C 180,E1 27500.632,E2 27500.632} C_VEL
LIN {X 0,Y 577.779,Z 792.334,A -85,B 0,C 180,E1 27499.668,E2 27499.668} C_VEL
LIN {X 0,Y 577.46,Z 810.442,A -85,B 0,C 180,E1 27498.531,E2 27498.531} C_VEL
LIN {X 0,Y 577.123,Z 827.816,A -85,B 0,C 180,E1 27497.224,E2 27497.224} C_VEL
LIN {X 0,Y 576.829,Z 843.538,A -85,B 0,C 180,E1 27495.828,E2 27495.828} C_VEL
LIN {X 0,Y 576.561,Z 858.636,A -85,B 0,C 180,E1 27494.257,E2 27494.257} C_VEL
LIN {X 0,Y 576.349,Z 872.401,A -85,B 0,C 180,E1 27492.572,E2 27492.572} C_VEL
LIN {X 0,Y 576.18,Z 885.136,A -85,B 0,C 180,E1 27490.725,E2 27490.725} C_VEL
LIN {X 0,Y 576.065,Z 895.554,A -85,B 0,C 180,E1 27488.921,E2 27488.921} C_VEL
LIN {X 0,Y 575.988,Z 904.694,A -85,B 0,C 180,E1 27487.011,E2 27487.011} C_VEL
LIN {X 0,Y 575.948,Z 912.406,A -85,B 0,C 180,E1 27484.974,E2 27484.974} C_VEL
LIN {X 0,Y 575.927,Z 918.047,A -85,B 0,C 180,E1 27483.014,E2 27483.014} C_VEL
LIN {X 0,Y 575.92,Z 922.296,A -85,B 0,C 180,E1 27480.92,E2 27480.92} C_VEL
LIN {X 0,Y 575.914,Z 924.733,A -85,B 0,C 180,E1 27478.855,E2 27478.855} C_VEL
LIN {X 0,Y 575.913,Z 925.477,A -85,B 0,C 180,E1 27476.827,E2 27476.827} C_VEL
LIN {X 0,Y 575.913,Z 924.512,A -85,B 0,C 180,E1 27474.731,E2 27474.731} C_VEL
LIN {X 0,Y 575.918,Z 921.782,A -85,B 0,C 180,E1 27472.667,E2 27472.667} C_VEL
LIN {X 0,Y 575.93,Z 917.381,A -85,B 0,C 180,E1 27470.633,E2 27470.633} C_VEL
LIN {X 0,Y 575.953,Z 911.164,A -85,B 0,C 180,E1 27468.583,E2 27468.583} C_VEL
LIN {X 0,Y 575.998,Z 903.453,A -85,B 0,C 180,E1 27466.623,E2 27466.623} C_VEL
LIN {X 0,Y 576.088,Z 894.478,A -85,B 0,C 180,E1 27464.779,E2 27464.779} C_VEL
LIN {X 0,Y 576.207,Z 883.551,A -85,B 0,C 180,E1 27462.932,E2 27462.932} C_VEL
LIN {X 0,Y 576.367,Z 871.367,A -85,B 0,C 180,E1 27461.201,E2 27461.201} C_VEL
LIN {X 0,Y 576.575,Z 857.984,A -85,B 0,C 180,E1 27459.581,E2 27459.581} C_VEL
LIN {X 0,Y 576.848,Z 842.334,A -85,B 0,C 180,E1 27457.968,E2 27457.968} C_VEL
LIN {X 0,Y 577.153,Z 825.41,A -85,B 0,C 180,E1 27456.495,E2 27456.495} C_VEL
LIN {X 0,Y 577.486,Z 807.948,A -85,B 0,C 180,E1 27455.213,E2 27455.213} C_VEL
LIN {X 0,Y 577.824,Z 790.141,A -85,B 0,C 180,E1 27454.116,E2 27454.116} C_VEL
LIN {X 0,Y 578.157,Z 770.355,A -85,B 0,C 180,E1 27453.121,E2 27453.121} C_VEL
LIN {X 0,Y 578.408,Z 751.053,A -85,B 0,C 180,E1 27452.351,E2 27452.351} C_VEL
LIN {X 0,Y 578.65,Z 730.738,A -85,B 0,C 180,E1 27451.737,E2 27451.737} C_VEL
LIN {X 0,Y 578.846,Z 709.593,A -85,B 0,C 180,E1 27451.297,E2 27451.297} C_VEL
LIN {X 0,Y 579.686,Z 457.972,A -85,B 0,C 180,E1 27447.882,E2 27447.882} C_VEL
LIN {X 0,Y 578.63,Z 452.06,A -85,B 0,C 180,E1 27447.72,E2 27447.72} C_VEL
LIN {X 0,Y 579.21,Z 409.869,A -85,B 0,C 180,E1 27444.6,E2 27444.6} C_VEL
LIN {X 0,Y 579.219,Z 402.708,A -85,B 0,C 180,E1 27444.053,E2 27444.053} C_VEL
LIN {X 0,Y 576.183,Z 394.177,A -85,B 0,C 180,E1 27443.156,E2 27443.156} C_VEL
LIN {X 0,Y 576.138,Z 393.964,A -85,B 0,C 180,E1 27440.004,E2 27440.004} C_VEL
LIN {X 0,Y 576.155,Z 393.961,A -85,B 0,C 180,E1 27436.654,E2 27436.654} C_VEL
LIN {X 0,Y 576.157,Z 393.959,A -85,B 0,C 180,E1 27433.324,E2 27433.324} C_VEL
LIN {X 0,Y 576.135,Z 393.967,A -85,B 0,C 180,E1 27430.007,E2 27430.007} C_VEL
LIN {X 0,Y 576.147,Z 393.955,A -85,B 0,C 180,E1 27426.799,E2 27426.799} C_VEL
LIN {X 0,Y 576.137,Z 393.963,A -85,B 0,C 180,E1 27423.51,E2 27423.51} C_VEL
LIN {X 0,Y 576.156,Z 393.971,A -85,B 0,C 180,E1 27420.193,E2 27420.193} C_VEL
LIN {X 0,Y 576.158,Z 393.96,A -85,B 0,C 180,E1 27416.861,E2 27416.861} C_VEL
LIN {X 0,Y 576.142,Z 393.968,A -85,B 0,C 180,E1 27413.592,E2 27413.592} C_VEL
LIN {X 0,Y 576.148,Z 393.959,A -85,B 0,C 180,E1 27410.402,E2 27410.402} C_VEL
LIN {X 0,Y 576.137,Z 393.963,A -85,B 0,C 180,E1 27407.231,E2 27407.231} C_VEL
LIN {X 0,Y 576.145,Z 393.964,A -85,B 0,C 180,E1 27404.071,E2 27404.071} C_VEL
LIN {X 0,Y 576.138,Z 393.963,A -85,B 0,C 180,E1 27400.829,E2 27400.829} C_VEL
LIN {X 0,Y 576.146,Z 393.966,A -85,B 0,C 180,E1 27397.653,E2 27397.653} C_VEL
LIN {X 0,Y 576.147,Z 393.961,A -85,B 0,C 180,E1 27394.334,E2 27394.334} C_VEL
LIN {X 0,Y 576.152,Z 393.967,A -85,B 0,C 180,E1 27390.91,E2 27390.91} C_VEL
LIN {X 0,Y 576.146,Z 393.962,A -85,B 0,C 180,E1 27387.604,E2 27387.604} C_VEL
LIN {X 0,Y 576.14,Z 393.964,A -85,B 0,C 180,E1 27384.34,E2 27384.34} C_VEL
LIN {X 0,Y 576.143,Z 393.964,A -85,B 0,C 180,E1 27381.16,E2 27381.16} C_VEL
LIN {X 0,Y 576.145,Z 393.962,A -85,B 0,C 180,E1 27377.889,E2 27377.889} C_VEL
LIN {X 0,Y 576.154,Z 393.967,A -85,B 0,C 180,E1 27374.574,E2 27374.574} C_VEL
LIN {X 0,Y 576.151,Z 393.961,A -85,B 0,C 180,E1 27371.208,E2 27371.208} C_VEL
LIN {X 0,Y 576.144,Z 393.965,A -85,B 0,C 180,E1 27367.88,E2 27367.88} C_VEL
LIN {X 0,Y 576.14,Z 393.964,A -85,B 0,C 180,E1 27364.679,E2 27364.679} C_VEL
LIN {X 0,Y 576.145,Z 393.963,A -85,B 0,C 180,E1 27361.392,E2 27361.392} C_VEL
LIN {X 0,Y 576.147,Z 393.966,A -85,B 0,C 180,E1 27358.111,E2 27358.111} C_VEL
LIN {X 0,Y 576.153,Z 393.96,A -85,B 0,C 180,E1 27354.723,E2 27354.723} C_VEL
LIN {X 0,Y 576.15,Z 393.968,A -85,B 0,C 180,E1 27351.417,E2 27351.417} C_VEL
LIN {X 0,Y 576.138,Z 393.962,A -85,B 0,C 180,E1 27348.181,E2 27348.181} C_VEL
LIN {X 0,Y 576.145,Z 393.964,A -85,B 0,C 180,E1 27344.912,E2 27344.912} C_VEL
LIN {X 0,Y 576.139,Z 393.966,A -85,B 0,C 180,E1 27341.676,E2 27341.676} C_VEL
LIN {X 0,Y 576.157,Z 393.959,A -85,B 0,C 180,E1 27338.307,E2 27338.307} C_VEL
LIN {X 0,Y 576.155,Z 393.968,A -85,B 0,C 180,E1 27334.943,E2 27334.943} C_VEL
LIN {X 0,Y 576.136,Z 393.963,A -85,B 0,C 180,E1 27331.628,E2 27331.628} C_VEL
LIN {X 0,Y 576.147,Z 393.964,A -85,B 0,C 180,E1 27328.441,E2 27328.441} C_VEL
LIN {X 0,Y 576.134,Z 393.966,A -85,B 0,C 180,E1 27325.173,E2 27325.173} C_VEL
LIN {X 0,Y 576.159,Z 393.961,A -85,B 0,C 180,E1 27321.826,E2 27321.826} C_VEL
LIN {X 0,Y 576.156,Z 393.971,A -85,B 0,C 180,E1 27318.415,E2 27318.415} C_VEL
LIN {X 0,Y 576.133,Z 393.959,A -85,B 0,C 180,E1 27315.063,E2 27315.063} C_VEL
LIN {X 0,Y 576.147,Z 393.954,A -85,B 0,C 180,E1 27311.885,E2 27311.885} C_VEL
LIN {X 0,Y 576.129,Z 393.939,A -85,B 0,C 180,E1 27308.651,E2 27308.651} C_VEL
LIN {X 0,Y 576.23,Z 394.479,A -85,B 0,C 180,E1 27308.268,E2 27308.268} C_VEL
LIN {X 0,Y 580.759,Z 404.923,A -85,B 0,C 180,E1 27307.226,E2 27307.226} C_VEL
LIN {X 0,Y 580.073,Z 455.205,A -85,B 0,C 180,E1 27304.134,E2 27304.134} C_VEL
LIN {X 0,Y 581.019,Z 462.223,A -85,B 0,C 180,E1 27303.965,E2 27303.965} C_VEL
LIN {X 0,Y 580.155,Z 682.632,A -85,B 0,C 180,E1 27300.855,E2 27300.855} C_VEL
LIN {X 0,Y 579.819,Z 761.965,A -85,B 0,C 180,E1 27299.728,E2 27299.728} C_VEL
LIN {X 0,Y 579.565,Z 783.201,A -85,B 0,C 180,E1 27299.24,E2 27299.24} C_VEL
LIN {X 0,Y 579.256,Z 804.715,A -85,B 0,C 180,E1 27298.565,E2 27298.565} C_VEL
LIN {X 0,Y 578.939,Z 825.096,A -85,B 0,C 180,E1 27297.74,E2 27297.74} C_VEL
LIN {X 0,Y 578.526,Z 844.721,A -85,B 0,C 180,E1 27296.759,E2 27296.759} C_VEL
LIN {X 0,Y 578.138,Z 864.696,A -85,B 0,C 180,E1 27295.564,E2 27295.564} C_VEL
LIN {X 0,Y 577.737,Z 883.811,A -85,B 0,C 180,E1 27294.21,E2 27294.21} C_VEL
LIN {X 0,Y 577.326,Z 901.673,A -85,B 0,C 180,E1 27292.72,E2 27292.72} C_VEL
LIN {X 0,Y 576.966,Z 918.824,A -85,B 0,C 180,E1 27291.059,E2 27291.059} C_VEL
LIN {X 0,Y 576.682,Z 934.155,A -85,B 0,C 180,E1 27289.341,E2 27289.341} C_VEL
LIN {X 0,Y 576.437,Z 948.613,A -85,B 0,C 180,E1 27287.464,E2 27287.464} C_VEL
LIN {X 0,Y 576.237,Z 960.82,A -85,B 0,C 180,E1 27285.603,E2 27285.603} C_VEL
LIN {X 0,Y 576.093,Z 972.282,A -85,B 0,C 180,E1 27283.552,E2 27283.552} C_VEL
LIN {X 0,Y 576.006,Z 981.836,A -85,B 0,C 180,E1 27281.517,E2 27281.517} C_VEL
LIN {X 0,Y 575.942,Z 989.523,A -85,B 0,C 180,E1 27279.495,E2 27279.495} C_VEL
LIN {X 0,Y 575.908,Z 995.886,A -85,B 0,C 180,E1 27277.383,E2 27277.383} C_VEL
LIN {X 0,Y 575.905,Z 1000.423,A -85,B 0,C 180,E1 27275.381,E2 27275.381} C_VEL
LIN {X 0,Y 575.911,Z 1003.557,A -85,B 0,C 180,E1 27273.286,E2 27273.286} C_VEL
LIN {X 0,Y 575.913,Z 1005.261,A -85,B 0,C 180,E1 27271.096,E2 27271.096} C_VEL
LIN {X 0,Y 575.905,Z 1005.285,A -85,B 0,C 180,E1 27269.007,E2 27269.007} C_VEL
LIN {X 0,Y 575.905,Z 1003.674,A -85,B 0,C 180,E1 27266.817,E2 27266.817} C_VEL
LIN {X 0,Y 575.9,Z 1000.636,A -85,B 0,C 180,E1 27264.723,E2 27264.723} C_VEL
LIN {X 0,Y 575.908,Z 996.15,A -85,B 0,C 180,E1 27262.721,E2 27262.721} C_VEL
LIN {X 0,Y 575.943,Z 989.893,A -85,B 0,C 180,E1 27260.61,E2 27260.61} C_VEL
LIN {X 0,Y 576.003,Z 982.668,A -85,B 0,C 180,E1 27258.691,E2 27258.691} C_VEL
LIN {X 0,Y 576.093,Z 973.343,A -85,B 0,C 180,E1 27256.657,E2 27256.657} C_VEL
LIN {X 0,Y 576.234,Z 962.756,A -85,B 0,C 180,E1 27254.71,E2 27254.71} C_VEL
LIN {X 0,Y 576.398,Z 950.765,A -85,B 0,C 180,E1 27252.852,E2 27252.852} C_VEL
LIN {X 0,Y 576.629,Z 936.741,A -85,B 0,C 180,E1 27250.978,E2 27250.978} C_VEL
LIN {X 0,Y 576.92,Z 921.66,A -85,B 0,C 180,E1 27249.237,E2 27249.237} C_VEL
LIN {X 0,Y 577.282,Z 904.76,A -85,B 0,C 180,E1 27247.554,E2 27247.554} C_VEL
LIN {X 0,Y 577.669,Z 886.494,A -85,B 0,C 180,E1 27246.002,E2 27246.002} C_VEL
LIN {X 0,Y 578.042,Z 867.987,A -85,B 0,C 180,E1 27244.656,E2 27244.656} C_VEL
LIN {X 0,Y 578.476,Z 848.783,A -85,B 0,C 180,E1 27243.465,E2 27243.465} C_VEL
LIN {X 0,Y 578.817,Z 829.865,A -85,B 0,C 180,E1 27242.482,E2 27242.482} C_VEL
LIN {X 0,Y 579.194,Z 808.523,A -85,B 0,C 180,E1 27241.577,E2 27241.577} C_VEL
LIN {X 0,Y 579.545,Z 787.407,A -85,B 0,C 180,E1 27240.874,E2 27240.874} C_VEL
LIN {X 0,Y 579.736,Z 766.488,A -85,B 0,C 180,E1 27240.363,E2 27240.363} C_VEL
LIN {X 0,Y 579.958,Z 737.747,A -85,B 0,C 180,E1 27239.909,E2 27239.909} C_VEL
LIN {X 0,Y 580.858,Z 503.893,A -85,B 0,C 180,E1 27236.631,E2 27236.631} C_VEL
LIN {X 0,Y 580.82,Z 459.51,A -85,B 0,C 180,E1 27235.983,E2 27235.983} C_VEL
LIN {X 0,Y 580.034,Z 454.156,A -85,B 0,C 180,E1 27235.813,E2 27235.813} C_VEL
LIN {X 0,Y 580.757,Z 405.056,A -85,B 0,C 180,E1 27232.782,E2 27232.782} C_VEL
LIN {X 0,Y 576.22,Z 394.45,A -85,B 0,C 180,E1 27231.727,E2 27231.727} C_VEL
LIN {X 0,Y 576.125,Z 393.94,A -85,B 0,C 180,E1 27231.349,E2 27231.349} C_VEL
LIN {X 0,Y 576.154,Z 393.963,A -85,B 0,C 180,E1 27228.115,E2 27228.115} C_VEL
LIN {X 0,Y 576.126,Z 393.966,A -85,B 0,C 180,E1 27224.926,E2 27224.926} C_VEL
LIN {X 0,Y 576.137,Z 393.971,A -85,B 0,C 180,E1 27221.59,E2 27221.59} C_VEL
LIN {X 0,Y 576.149,Z 393.964,A -85,B 0,C 180,E1 27218.34,E2 27218.34} C_VEL
LIN {X 0,Y 576.106,Z 393.969,A -85,B 0,C 180,E1 27215.062,E2 27215.062} C_VEL
LIN {X 0,Y 576.161,Z 393.969,A -85,B 0,C 180,E1 27211.84,E2 27211.84} C_VEL
LIN {X 0,Y 576.095,Z 393.968,A -85,B 0,C 180,E1 27208.734,E2 27208.734} C_VEL
LIN {X 0,Y 576.147,Z 393.971,A -85,B 0,C 180,E1 27205.531,E2 27205.531} C_VEL
LIN {X 0,Y 576.086,Z 393.97,A -85,B 0,C 180,E1 27202.555,E2 27202.555} C_VEL
LIN {X 0,Y 576.132,Z 393.971,A -85,B 0,C 180,E1 27199.358,E2 27199.358} C_VEL
LIN {X 0,Y 576.077,Z 393.971,A -85,B 0,C 180,E1 27196.314,E2 27196.314} C_VEL
LIN {X 0,Y 576.103,Z 393.971,A -85,B 0,C 180,E1 27193.039,E2 27193.039} C_VEL
LIN {X 0,Y 576.084,Z 393.971,A -85,B 0,C 180,E1 27190.096,E2 27190.096} C_VEL
LIN {X 0,Y 576.105,Z 393.969,A -85,B 0,C 180,E1 27186.777,E2 27186.777} C_VEL
LIN {X 0,Y 576.107,Z 393.97,A -85,B 0,C 180,E1 27183.781,E2 27183.781} C_VEL
LIN {X 0,Y 576.104,Z 393.968,A -85,B 0,C 180,E1 27180.497,E2 27180.497} C_VEL
LIN {X 0,Y 576.14,Z 393.971,A -85,B 0,C 180,E1 27177.414,E2 27177.414} C_VEL
LIN {X 0,Y 576.106,Z 393.967,A -85,B 0,C 180,E1 27174.122,E2 27174.122} C_VEL
LIN {X 0,Y 576.161,Z 393.967,A -85,B 0,C 180,E1 27170.914,E2 27170.914} C_VEL
LIN {X 0,Y 576.117,Z 393.968,A -85,B 0,C 180,E1 27167.674,E2 27167.674} C_VEL
LIN {X 0,Y 576.151,Z 393.963,A -85,B 0,C 180,E1 27164.383,E2 27164.383} C_VEL
LIN {X 0,Y 576.145,Z 393.97,A -85,B 0,C 180,E1 27163.244,E2 27163.244} C_VEL
LIN {X 0,Y 575.185,Z 394.097,A -85,B 0,C 180,E1 27162.478,E2 27162.478} C_VEL
LIN {X 0,Y 568.732,Z 394.889,A -85,B 0,C 180,E1 27160.327,E2 27160.327} C_VEL
LIN {X 0,Y 568.188,Z 394.956,A -85,B 0,C 180,E1 27159.767,E2 27159.767} C_VEL
LIN {X 0,Y 568.214,Z 394.956,A -85,B 0,C 180,E1 27156.566,E2 27156.566} C_VEL
LIN {X 0,Y 568.203,Z 394.956,A -85,B 0,C 180,E1 27153.225,E2 27153.225} C_VEL
LIN {X 0,Y 568.237,Z 395.192,A -85,B 0,C 180,E1 27151.218,E2 27151.218} C_VEL
LIN {X 0,Y 570.23,Z 400.761,A -85,B 0,C 180,E1 27150.596,E2 27150.596} C_VEL
LIN {X 0,Y 572.169,Z 406.572,A -85,B 0,C 180,E1 27150.014,E2 27150.014} C_VEL
LIN {X 0,Y 571.404,Z 449.366,A -85,B 0,C 180,E1 27146.791,E2 27146.791} C_VEL
LIN {X 0,Y 571.5,Z 453.107,A -85,B 0,C 180,E1 27146.557,E2 27146.557} C_VEL
LIN {X 0,Y 572.681,Z 460.586,A -85,B 0,C 180,E1 27146.382,E2 27146.382} C_VEL
LIN {X 0,Y 571.615,Z 713.859,A -85,B 0,C 180,E1 27142.892,E2 27142.892} C_VEL
LIN {X 0,Y 571.356,Z 734.373,A -85,B 0,C 180,E1 27142.421,E2 27142.421} C_VEL
LIN {X 0,Y 571.033,Z 753.821,A -85,B 0,C 180,E1 27141.794,E2 27141.794} C_VEL
LIN {X 0,Y 570.672,Z 773.703,A -85,B 0,C 180,E1 27140.959,E2 27140.959} C_VEL
LIN {X 0,Y 570.297,Z 791.968,A -85,B 0,C 180,E1 27140.005,E2 27140.005} C_VEL
LIN {X 0,Y 569.875,Z 810.648,A -85,B 0,C 180,E1 27138.819,E2 27138.819} C_VEL
LIN {X 0,Y 569.449,Z 828.322,A -85,B 0,C 180,E1 27137.468,E2 27137.468} C_VEL
LIN {X 0,Y 569.065,Z 844.845,A -85,B 0,C 180,E1 27135.969,E2 27135.969} C_VEL
LIN {X 0,Y 568.733,Z 859.55,A -85,B 0,C 180,E1 27134.398,E2 27134.398} C_VEL
LIN {X 0,Y 568.462,Z 873.292,A -85,B 0,C 180,E1 27132.674,E2 27132.674} C_VEL
LIN {X 0,Y 568.255,Z 885.666,A -85,B 0,C 180,E1 27130.835,E2 27130.835} C_VEL
LIN {X 0,Y 568.093,Z 896.672,A -85,B 0,C 180,E1 27128.87,E2 27128.87} C_VEL
LIN {X 0,Y 568,Z 905.517,A -85,B 0,C 180,E1 27126.947,E2 27126.947} C_VEL
LIN {X 0,Y 567.957,Z 912.645,A -85,B 0,C 180,E1 27125.019,E2 27125.019} C_VEL
LIN {X 0,Y 567.93,Z 918.125,A -85,B 0,C 180,E1 27123.069,E2 27123.069} C_VEL
LIN {X 0,Y 567.919,Z 922.299,A -85,B 0,C 180,E1 27120.974,E2 27120.974} C_VEL
LIN {X 0,Y 567.914,Z 924.762,A -85,B 0,C 180,E1 27118.839,E2 27118.839} C_VEL
LIN {X 0,Y 567.912,Z 925.468,A -85,B 0,C 180,E1 27116.786,E2 27116.786} C_VEL
LIN {X 0,Y 567.911,Z 924.476,A -85,B 0,C 180,E1 27114.658,E2 27114.658} C_VEL
LIN {X 0,Y 567.917,Z 921.719,A -85,B 0,C 180,E1 27112.566,E2 27112.566} C_VEL
LIN {X 0,Y 567.932,Z 917.555,A -85,B 0,C 180,E1 27110.613,E2 27110.613} C_VEL
LIN {X 0,Y 567.964,Z 911.189,A -85,B 0,C 180,E1 27108.471,E2 27108.471} C_VEL
LIN {X 0,Y 568.028,Z 903.379,A -85,B 0,C 180,E1 27106.46,E2 27106.46} C_VEL
LIN {X 0,Y 568.143,Z 894.169,A -85,B 0,C 180,E1 27104.549,E2 27104.549} C_VEL
LIN {X 0,Y 568.305,Z 882.722,A -85,B 0,C 180,E1 27102.598,E2 27102.598} C_VEL
LIN {X 0,Y 568.528,Z 870.378,A -85,B 0,C 180,E1 27100.844,E2 27100.844} C_VEL
LIN {X 0,Y 568.797,Z 856.818,A -85,B 0,C 180,E1 27099.202,E2 27099.202} C_VEL
LIN {X 0,Y 569.142,Z 841.491,A -85,B 0,C 180,E1 27097.62,E2 27097.62} C_VEL
LIN {X 0,Y 569.528,Z 824.642,A -85,B 0,C 180,E1 27096.145,E2 27096.145} C_VEL
LIN {X 0,Y 569.944,Z 806.715,A -85,B 0,C 180,E1 27094.827,E2 27094.827} C_VEL
LIN {X 0,Y 570.352,Z 788.644,A -85,B 0,C 180,E1 27093.717,E2 27093.717} C_VEL
LIN {X 0,Y 570.778,Z 769.644,A -85,B 0,C 180,E1 27092.759,E2 27092.759} C_VEL
LIN {X 0,Y 571.114,Z 750.068,A -85,B 0,C 180,E1 27091.979,E2 27091.979} C_VEL
LIN {X 0,Y 571.393,Z 729.979,A -85,B 0,C 180,E1 27091.373,E2 27091.373} C_VEL
LIN {X 0,Y 571.633,Z 708.874,A -85,B 0,C 180,E1 27090.937,E2 27090.937} C_VEL
LIN {X 0,Y 572.687,Z 459.39,A -85,B 0,C 180,E1 27087.512,E2 27087.512} C_VEL
LIN {X 0,Y 571.388,Z 452.341,A -85,B 0,C 180,E1 27087.328,E2 27087.328} C_VEL
LIN {X 0,Y 572.099,Z 410.292,A -85,B 0,C 180,E1 27084.18,E2 27084.18} C_VEL
LIN {X 0,Y 572.049,Z 405.789,A -85,B 0,C 180,E1 27083.827,E2 27083.827} C_VEL
LIN {X 0,Y 568.252,Z 395.281,A -85,B 0,C 180,E1 27082.72,E2 27082.72} C_VEL
LIN {X 0,Y 568.213,Z 394.943,A -85,B 0,C 180,E1 27081.467,E2 27081.467} C_VEL
LIN {X 0,Y 568.193,Z 394.952,A -85,B 0,C 180,E1 27078.22,E2 27078.22} C_VEL
LIN {X 0,Y 568.211,Z 394.956,A -85,B 0,C 180,E1 27075.007,E2 27075.007} C_VEL
LIN {X 0,Y 568.199,Z 394.949,A -85,B 0,C 180,E1 27071.745,E2 27071.745} C_VEL
LIN {X 0,Y 568.22,Z 394.948,A -85,B 0,C 180,E1 27068.421,E2 27068.421} C_VEL
LIN {X 0,Y 568.214,Z 394.95,A -85,B 0,C 180,E1 27064.989,E2 27064.989} C_VEL
LIN {X 0,Y 568.198,Z 394.956,A -85,B 0,C 180,E1 27061.746,E2 27061.746} C_VEL
LIN {X 0,Y 568.207,Z 394.952,A -85,B 0,C 180,E1 27058.49,E2 27058.49} C_VEL
LIN {X 0,Y 568.198,Z 394.949,A -85,B 0,C 180,E1 27055.238,E2 27055.238} C_VEL
LIN {X 0,Y 568.221,Z 394.956,A -85,B 0,C 180,E1 27051.855,E2 27051.855} C_VEL
LIN {X 0,Y 568.214,Z 394.951,A -85,B 0,C 180,E1 27048.44,E2 27048.44} C_VEL
LIN {X 0,Y 568.199,Z 394.954,A -85,B 0,C 180,E1 27045.118,E2 27045.118} C_VEL
LIN {X 0,Y 568.208,Z 394.953,A -85,B 0,C 180,E1 27041.83,E2 27041.83} C_VEL
LIN {X 0,Y 568.208,Z 394.95,A -85,B 0,C 180,E1 27038.53,E2 27038.53} C_VEL
LIN {X 0,Y 568.211,Z 394.959,A -85,B 0,C 180,E1 27035.09,E2 27035.09} C_VEL
LIN {X 0,Y 568.207,Z 394.949,A -85,B 0,C 180,E1 27031.746,E2 27031.746} C_VEL
LIN {X 0,Y 568.2,Z 394.954,A -85,B 0,C 180,E1 27028.482,E2 27028.482} C_VEL
LIN {X 0,Y 568.205,Z 394.95,A -85,B 0,C 180,E1 27025.204,E2 27025.204} C_VEL
LIN {X 0,Y 568.212,Z 394.949,A -85,B 0,C 180,E1 27021.904,E2 27021.904} C_VEL
LIN {X 0,Y 568.213,Z 394.958,A -85,B 0,C 180,E1 27018.466,E2 27018.466} C_VEL
LIN {X 0,Y 568.206,Z 394.949,A -85,B 0,C 180,E1 27015.2,E2 27015.2} C_VEL
LIN {X 0,Y 568.203,Z 394.954,A -85,B 0,C 180,E1 27011.882,E2 27011.882} C_VEL
LIN {X 0,Y 568.204,Z 394.952,A -85,B 0,C 180,E1 27008.602,E2 27008.602} C_VEL
LIN {X 0,Y 568.216,Z 394.949,A -85,B 0,C 180,E1 27005.25,E2 27005.25} C_VEL
LIN {X 0,Y 568.211,Z 394.957,A -85,B 0,C 180,E1 27001.815,E2 27001.815} C_VEL
LIN {X 0,Y 568.201,Z 394.951,A -85,B 0,C 180,E1 26998.488,E2 26998.488} C_VEL
LIN {X 0,Y 568.205,Z 394.953,A -85,B 0,C 180,E1 26995.256,E2 26995.256} C_VEL
LIN {X 0,Y 568.201,Z 394.951,A -85,B 0,C 180,E1 26992.009,E2 26992.009} C_VEL
LIN {X 0,Y 568.219,Z 394.947,A -85,B 0,C 180,E1 26988.634,E2 26988.634} C_VEL
LIN {X 0,Y 568.212,Z 394.956,A -85,B 0,C 180,E1 26985.218,E2 26985.218} C_VEL
LIN {X 0,Y 568.199,Z 394.952,A -85,B 0,C 180,E1 26981.959,E2 26981.959} C_VEL
LIN {X 0,Y 568.208,Z 394.953,A -85,B 0,C 180,E1 26978.747,E2 26978.747} C_VEL
LIN {X 0,Y 568.198,Z 394.955,A -85,B 0,C 180,E1 26975.474,E2 26975.474} C_VEL
LIN {X 0,Y 568.22,Z 394.948,A -85,B 0,C 180,E1 26972.092,E2 26972.092} C_VEL
LIN {X 0,Y 568.219,Z 394.955,A -85,B 0,C 180,E1 26968.729,E2 26968.729} C_VEL
LIN {X 0,Y 568.197,Z 394.953,A -85,B 0,C 180,E1 26965.442,E2 26965.442} C_VEL
LIN {X 0,Y 568.21,Z 394.955,A -85,B 0,C 180,E1 26962.195,E2 26962.195} C_VEL
LIN {X 0,Y 568.195,Z 394.953,A -85,B 0,C 180,E1 26958.977,E2 26958.977} C_VEL
LIN {X 0,Y 568.214,Z 394.943,A -85,B 0,C 180,E1 26955.687,E2 26955.687} C_VEL
LIN {X 0,Y 568.213,Z 394.944,A -85,B 0,C 180,E1 26952.349,E2 26952.349} C_VEL
LIN {X 0,Y 568.217,Z 395.092,A -85,B 0,C 180,E1 26948.944,E2 26948.944} C_VEL
LIN {X 0,Y 568.431,Z 396.119,A -85,B 0,C 180,E1 26948.771,E2 26948.771} C_VEL
LIN {X 0,Y 573.995,Z 408.757,A -85,B 0,C 180,E1 26947.491,E2 26947.491} C_VEL
LIN {X 0,Y 573.251,Z 455.659,A -85,B 0,C 180,E1 26944.588,E2 26944.588} C_VEL
LIN {X 0,Y 574.374,Z 463.49,A -85,B 0,C 180,E1 26944.393,E2 26944.393} C_VEL
LIN {X 0,Y 573.281,Z 683.973,A -85,B 0,C 180,E1 26941.247,E2 26941.247} C_VEL
LIN {X 0,Y 572.865,Z 762.072,A -85,B 0,C 180,E1 26940.124,E2 26940.124} C_VEL
LIN {X 0,Y 572.543,Z 783.461,A -85,B 0,C 180,E1 26939.627,E2 26939.627} C_VEL
LIN {X 0,Y 572.144,Z 805.567,A -85,B 0,C 180,E1 26938.92,E2 26938.92} C_VEL
LIN {X 0,Y 571.738,Z 826.359,A -85,B 0,C 180,E1 26938.064,E2 26938.064} C_VEL
LIN {X 0,Y 571.205,Z 846.491,A -85,B 0,C 180,E1 26937.03,E2 26937.03} C_VEL
LIN {X 0,Y 570.672,Z 867.117,A -85,B 0,C 180,E1 26935.756,E2 26935.756} C_VEL
LIN {X 0,Y 570.179,Z 885.766,A -85,B 0,C 180,E1 26934.393,E2 26934.393} C_VEL
LIN {X 0,Y 569.683,Z 903.647,A -85,B 0,C 180,E1 26932.864,E2 26932.864} C_VEL
LIN {X 0,Y 569.236,Z 920.177,A -85,B 0,C 180,E1 26931.215,E2 26931.215} C_VEL
LIN {X 0,Y 568.86,Z 935.856,A -85,B 0,C 180,E1 26929.404,E2 26929.404} C_VEL
LIN {X 0,Y 568.554,Z 950.029,A -85,B 0,C 180,E1 26927.503,E2 26927.503} C_VEL
LIN {X 0,Y 568.318,Z 962.727,A -85,B 0,C 180,E1 26925.512,E2 26925.512} C_VEL
LIN {X 0,Y 568.139,Z 973.322,A -85,B 0,C 180,E1 26923.538,E2 26923.538} C_VEL
LIN {X 0,Y 568.025,Z 983.152,A -85,B 0,C 180,E1 26921.349,E2 26921.349} C_VEL
LIN {X 0,Y 567.96,Z 990.93,A -85,B 0,C 180,E1 26919.22,E2 26919.22} C_VEL
LIN {X 0,Y 567.913,Z 996.648,A -85,B 0,C 180,E1 26917.183,E2 26917.183} C_VEL
LIN {X 0,Y 567.895,Z 1001.142,A -85,B 0,C 180,E1 26915.052,E2 26915.052} C_VEL
LIN {X 0,Y 567.896,Z 1003.894,A -85,B 0,C 180,E1 26913.03,E2 26913.03} C_VEL
LIN {X 0,Y 567.898,Z 1005.328,A -85,B 0,C 180,E1 26910.809,E2 26910.809} C_VEL
LIN {X 0,Y 567.906,Z 1005.21,A -85,B 0,C 180,E1 26908.691,E2 26908.691} C_VEL
LIN {X 0,Y 567.914,Z 1003.449,A -85,B 0,C 180,E1 26906.571,E2 26906.571} C_VEL
LIN {X 0,Y 567.921,Z 1000.019,A -85,B 0,C 180,E1 26904.344,E2 26904.344} C_VEL
LIN {X 0,Y 567.929,Z 995.388,A -85,B 0,C 180,E1 26902.313,E2 26902.313} C_VEL
LIN {X 0,Y 567.964,Z 988.829,A -85,B 0,C 180,E1 26900.17,E2 26900.17} C_VEL
LIN {X 0,Y 568.045,Z 980.991,A -85,B 0,C 180,E1 26898.118,E2 26898.118} C_VEL
LIN {X 0,Y 568.156,Z 971.786,A -85,B 0,C 180,E1 26896.155,E2 26896.155} C_VEL
LIN {X 0,Y 568.341,Z 960.207,A -85,B 0,C 180,E1 26894.074,E2 26894.074} C_VEL
LIN {X 0,Y 568.597,Z 947.898,A -85,B 0,C 180,E1 26892.186,E2 26892.186} C_VEL
LIN {X 0,Y 568.928,Z 933.342,A -85,B 0,C 180,E1 26890.283,E2 26890.283} C_VEL
LIN {X 0,Y 569.304,Z 918.076,A -85,B 0,C 180,E1 26888.564,E2 26888.564} C_VEL
LIN {X 0,Y 569.758,Z 900.518,A -85,B 0,C 180,E1 26886.856,E2 26886.856} C_VEL
LIN {X 0,Y 570.243,Z 883.066,A -85,B 0,C 180,E1 26885.394,E2 26885.394} C_VEL
LIN {X 0,Y 570.778,Z 863.953,A -85,B 0,C 180,E1 26884.031,E2 26884.031} C_VEL
LIN {X 0,Y 571.247,Z 844.811,A -85,B 0,C 180,E1 26882.877,E2 26882.877} C_VEL
LIN {X 0,Y 571.756,Z 825.208,A -85,B 0,C 180,E1 26881.885,E2 26881.885} C_VEL
LIN {X 0,Y 572.166,Z 804.843,A -85,B 0,C 180,E1 26881.053,E2 26881.053} C_VEL
LIN {X 0,Y 572.548,Z 782.738,A -85,B 0,C 180,E1 26880.353,E2 26880.353} C_VEL
LIN {X 0,Y 572.87,Z 761.296,A -85,B 0,C 180,E1 26879.863,E2 26879.863} C_VEL
LIN {X 0,Y 573.631,Z 608.695,A -85,B 0,C 180,E1 26877.688,E2 26877.688} C_VEL
LIN {X 0,Y 574.223,Z 461.202,A -85,B 0,C 180,E1 26875.562,E2 26875.562} C_VEL
LIN {X 0,Y 573.151,Z 454.156,A -85,B 0,C 180,E1 26875.344,E2 26875.344} C_VEL
LIN {X 0,Y 573.986,Z 408.469,A -85,B 0,C 180,E1 26872.489,E2 26872.489} C_VEL
LIN {X 0,Y 568.253,Z 395.352,A -85,B 0,C 180,E1 26871.142,E2 26871.142} C_VEL
LIN {X 0,Y 568.219,Z 394.94,A -85,B 0,C 180,E1 26870.698,E2 26870.698} C_VEL
LIN {X 0,Y 568.186,Z 394.959,A -85,B 0,C 180,E1 26867.355,E2 26867.355} C_VEL
LIN {X 0,Y 568.219,Z 394.958,A -85,B 0,C 180,E1 26864.121,E2 26864.121} C_VEL
LIN {X 0,Y 568.181,Z 394.956,A -85,B 0,C 180,E1 26860.891,E2 26860.891} C_VEL
LIN {X 0,Y 568.205,Z 394.96,A -85,B 0,C 180,E1 26857.633,E2 26857.633} C_VEL
LIN {X 0,Y 568.182,Z 394.955,A -85,B 0,C 180,E1 26854.516,E2 26854.516} C_VEL
LIN {X 0,Y 568.169,Z 394.959,A -85,B 0,C 180,E1 26851.156,E2 26851.156} C_VEL
LIN {X 0,Y 568.208,Z 394.955,A -85,B 0,C 180,E1 26848.023,E2 26848.023} C_VEL
LIN {X 0,Y 568.15,Z 394.958,A -85,B 0,C 180,E1 26844.767,E2 26844.767} C_VEL
LIN {X 0,Y 568.218,Z 394.958,A -85,B 0,C 180,E1 26841.578,E2 26841.578} C_VEL
LIN {X 0,Y 568.14,Z 394.959,A -85,B 0,C 180,E1 26838.467,E2 26838.467} C_VEL
LIN {X 0,Y 568.19,Z 394.958,A -85,B 0,C 180,E1 26835.305,E2 26835.305} C_VEL
LIN {X 0,Y 568.14,Z 394.96,A -85,B 0,C 180,E1 26832.192,E2 26832.192} C_VEL
LIN {X 0,Y 568.169,Z 394.956,A -85,B 0,C 180,E1 26828.908,E2 26828.908} C_VEL
LIN {X 0,Y 568.155,Z 394.96,A -85,B 0,C 180,E1 26825.959,E2 26825.959} C_VEL
LIN {X 0,Y 568.161,Z 394.956,A -85,B 0,C 180,E1 26822.521,E2 26822.521} C_VEL
LIN {X 0,Y 568.206,Z 394.959,A -85,B 0,C 180,E1 26819.395,E2 26819.395} C_VEL
LIN {X 0,Y 568.164,Z 394.955,A -85,B 0,C 180,E1 26816.148,E2 26816.148} C_VEL
LIN {X 0,Y 568.223,Z 394.955,A -85,B 0,C 180,E1 26812.912,E2 26812.912} C_VEL
LIN {X 0,Y 568.178,Z 394.958,A -85,B 0,C 180,E1 26809.659,E2 26809.659} C_VEL
LIN {X 0,Y 568.203,Z 394.952,A -85,B 0,C 180,E1 26806.361,E2 26806.361} C_VEL
LIN {X 0,Y 568.214,Z 394.961,A -85,B 0,C 180,E1 26803.121,E2 26803.121} C_VEL
LIN {X 0,Y 568.19,Z 394.956,A -85,B 0,C 180,E1 26799.824,E2 26799.824} C_VEL
LIN {X 0,Y 568.188,Z 394.956,A -85,B 0,C 180,E1 26799.767,E2 26799.767} C_VEL
LIN {X 0,Y 567.2,Z 395.083,A -85,B 0,C 180,E1 26798.991,E2 26798.991} C_VEL
LIN {X 0,Y 560.818,Z 395.881,A -85,B 0,C 180,E1 26796.81,E2 26796.81} C_VEL
LIN {X 0,Y 560.282,Z 395.941,A -85,B 0,C 180,E1 26796.242,E2 26796.242} C_VEL
LIN {X 0,Y 560.276,Z 395.937,A -85,B 0,C 180,E1 26792.815,E2 26792.815} C_VEL
LIN {X 0,Y 560.3,Z 396.211,A -85,B 0,C 180,E1 26791.719,E2 26791.719} C_VEL
LIN {X 0,Y 563.653,Z 405.233,A -85,B 0,C 180,E1 26790.686,E2 26790.686} C_VEL
LIN {X 0,Y 565.041,Z 409.674,A -85,B 0,C 180,E1 26790.241,E2 26790.241} C_VEL
LIN {X 0,Y 564.147,Z 451.779,A -85,B 0,C 180,E1 26787.036,E2 26787.036} C_VEL
LIN {X 0,Y 565.615,Z 460.134,A -85,B 0,C 180,E1 26786.793,E2 26786.793} C_VEL
LIN {X 0,Y 564.674,Z 667.633,A -85,B 0,C 180,E1 26783.908,E2 26783.908} C_VEL
LIN {X 0,Y 564.389,Z 715.221,A -85,B 0,C 180,E1 26783.222,E2 26783.222} C_VEL
LIN {X 0,Y 564.09,Z 736.055,A -85,B 0,C 180,E1 26782.727,E2 26782.727} C_VEL
LIN {X 0,Y 563.683,Z 756.287,A -85,B 0,C 180,E1 26782.046,E2 26782.046} C_VEL
LIN {X 0,Y 563.226,Z 775.791,A -85,B 0,C 180,E1 26781.193,E2 26781.193} C_VEL
LIN {X 0,Y 562.729,Z 795.241,A -85,B 0,C 180,E1 26780.131,E2 26780.131} C_VEL
LIN {X 0,Y 562.217,Z 813.713,A -85,B 0,C 180,E1 26778.903,E2 26778.903} C_VEL
LIN {X 0,Y 561.737,Z 830.449,A -85,B 0,C 180,E1 26777.577,E2 26777.577} C_VEL
LIN {X 0,Y 561.3,Z 846.233,A -85,B 0,C 180,E1 26776.105,E2 26776.105} C_VEL
LIN {X 0,Y 560.894,Z 861.124,A -85,B 0,C 180,E1 26774.468,E2 26774.468} C_VEL
LIN {X 0,Y 560.565,Z 874.728,A -85,B 0,C 180,E1 26772.703,E2 26772.703} C_VEL
LIN {X 0,Y 560.324,Z 886.445,A -85,B 0,C 180,E1 26770.907,E2 26770.907} C_VEL
LIN {X 0,Y 560.131,Z 897.261,A -85,B 0,C 180,E1 26768.923,E2 26768.923} C_VEL
LIN {X 0,Y 560.012,Z 906.427,A -85,B 0,C 180,E1 26766.859,E2 26766.859} C_VEL
LIN {X 0,Y 559.959,Z 913.534,A -85,B 0,C 180,E1 26764.843,E2 26764.843} C_VEL
LIN {X 0,Y 559.929,Z 919.12,A -85,B 0,C 180,E1 26762.747,E2 26762.747} C_VEL
LIN {X 0,Y 559.915,Z 922.798,A -85,B 0,C 180,E1 26760.708,E2 26760.708} C_VEL
LIN {X 0,Y 559.908,Z 924.866,A -85,B 0,C 180,E1 26758.706,E2 26758.706} C_VEL
LIN {X 0,Y 559.905,Z 925.434,A -85,B 0,C 180,E1 26756.627,E2 26756.627} C_VEL
LIN {X 0,Y 559.911,Z 924.434,A -85,B 0,C 180,E1 26754.584,E2 26754.584} C_VEL
LIN {X 0,Y 559.918,Z 921.656,A -85,B 0,C 180,E1 26752.463,E2 26752.463} C_VEL
LIN {X 0,Y 559.935,Z 917.461,A -85,B 0,C 180,E1 26750.484,E2 26750.484} C_VEL
LIN {X 0,Y 559.976,Z 911.433,A -85,B 0,C 180,E1 26748.421,E2 26748.421} C_VEL
LIN {X 0,Y 560.048,Z 904.17,A -85,B 0,C 180,E1 26746.488,E2 26746.488} C_VEL
LIN {X 0,Y 560.188,Z 894.683,A -85,B 0,C 180,E1 26744.468,E2 26744.468} C_VEL
LIN {X 0,Y 560.373,Z 883.811,A -85,B 0,C 180,E1 26742.57,E2 26742.57} C_VEL
LIN {X 0,Y 560.638,Z 871.686,A -85,B 0,C 180,E1 26740.79,E2 26740.79} C_VEL
LIN {X 0,Y 560.986,Z 857.462,A -85,B 0,C 180,E1 26739.021,E2 26739.021} C_VEL
LIN {X 0,Y 561.42,Z 841.717,A -85,B 0,C 180,E1 26737.365,E2 26737.365} C_VEL
LIN {X 0,Y 561.887,Z 825.108,A -85,B 0,C 180,E1 26735.887,E2 26735.887} C_VEL
LIN {X 0,Y 562.377,Z 807.793,A -85,B 0,C 180,E1 26734.587,E2 26734.587} C_VEL
LIN {X 0,Y 562.873,Z 789.918,A -85,B 0,C 180,E1 26733.46,E2 26733.46} C_VEL
LIN {X 0,Y 563.394,Z 770.009,A -85,B 0,C 180,E1 26732.439,E2 26732.439} C_VEL
LIN {X 0,Y 563.807,Z 750.494,A -85,B 0,C 180,E1 26731.649,E2 26731.649} C_VEL
LIN {X 0,Y 564.148,Z 730.293,A -85,B 0,C 180,E1 26731.029,E2 26731.029} C_VEL
LIN {X 0,Y 564.438,Z 709.129,A -85,B 0,C 180,E1 26730.585,E2 26730.585} C_VEL
LIN {X 0,Y 565.713,Z 460.634,A -85,B 0,C 180,E1 26727.13,E2 26727.13} C_VEL
LIN {X 0,Y 564.152,Z 452.166,A -85,B 0,C 180,E1 26726.899,E2 26726.899} C_VEL
LIN {X 0,Y 565.033,Z 410.059,A -85,B 0,C 180,E1 26723.699,E2 26723.699} C_VEL
LIN {X 0,Y 563.986,Z 406.277,A -85,B 0,C 180,E1 26723.33,E2 26723.33} C_VEL
LIN {X 0,Y 560.292,Z 396.204,A -85,B 0,C 180,E1 26722.203,E2 26722.203} C_VEL
LIN {X 0,Y 560.273,Z 395.945,A -85,B 0,C 180,E1 26719.198,E2 26719.198} C_VEL
LIN {X 0,Y 560.258,Z 395.943,A -85,B 0,C 180,E1 26715.952,E2 26715.952} C_VEL
LIN {X 0,Y 560.277,Z 395.933,A -85,B 0,C 180,E1 26712.552,E2 26712.552} C_VEL
LIN {X 0,Y 560.278,Z 395.94,A -85,B 0,C 180,E1 26709.197,E2 26709.197} C_VEL
LIN {X 0,Y 560.259,Z 395.943,A -85,B 0,C 180,E1 26705.876,E2 26705.876} C_VEL
LIN {X 0,Y 560.271,Z 395.944,A -85,B 0,C 180,E1 26702.584,E2 26702.584} C_VEL
LIN {X 0,Y 560.262,Z 395.938,A -85,B 0,C 180,E1 26699.308,E2 26699.308} C_VEL
LIN {X 0,Y 560.275,Z 395.944,A -85,B 0,C 180,E1 26695.899,E2 26695.899} C_VEL
LIN {X 0,Y 560.272,Z 395.941,A -85,B 0,C 180,E1 26692.514,E2 26692.514} C_VEL
LIN {X 0,Y 560.26,Z 395.943,A -85,B 0,C 180,E1 26689.217,E2 26689.217} C_VEL
LIN {X 0,Y 560.27,Z 395.94,A -85,B 0,C 180,E1 26685.892,E2 26685.892} C_VEL
LIN {X 0,Y 560.274,Z 395.936,A -85,B 0,C 180,E1 26682.519,E2 26682.519} C_VEL
LIN {X 0,Y 560.272,Z 395.946,A -85,B 0,C 180,E1 26679.18,E2 26679.18} C_VEL
LIN {X 0,Y 560.267,Z 395.937,A -85,B 0,C 180,E1 26675.828,E2 26675.828} C_VEL
LIN {X 0,Y 560.262,Z 395.94,A -85,B 0,C 180,E1 26672.61,E2 26672.61} C_VEL
LIN {X 0,Y 560.27,Z 395.943,A -85,B 0,C 180,E1 26669.274,E2 26669.274} C_VEL
LIN {X 0,Y 560.276,Z 395.932,A -85,B 0,C 180,E1 26665.916,E2 26665.916} C_VEL
LIN {X 0,Y 560.273,Z 395.945,A -85,B 0,C 180,E1 26662.563,E2 26662.563} C_VEL
LIN {X 0,Y 560.265,Z 395.937,A -85,B 0,C 180,E1 26659.253,E2 26659.253} C_VEL
LIN {X 0,Y 560.264,Z 395.939,A -85,B 0,C 180,E1 26655.952,E2 26655.952} C_VEL
LIN {X 0,Y 560.268,Z 395.943,A -85,B 0,C 180,E1 26652.68,E2 26652.68} C_VEL
LIN {X 0,Y 560.276,Z 395.934,A -85,B 0,C 180,E1 26649.243,E2 26649.243} C_VEL
LIN {X 0,Y 560.272,Z 395.945,A -85,B 0,C 180,E1 26645.941,E2 26645.941} C_VEL
LIN {X 0,Y 560.262,Z 395.936,A -85,B 0,C 180,E1 26642.66,E2 26642.66} C_VEL
LIN {X 0,Y 560.266,Z 395.939,A -85,B 0,C 180,E1 26639.387,E2 26639.387} C_VEL
LIN {X 0,Y 560.269,Z 395.944,A -85,B 0,C 180,E1 26636.03,E2 26636.03} C_VEL
LIN {X 0,Y 560.274,Z 395.933,A -85,B 0,C 180,E1 26632.618,E2 26632.618} C_VEL
LIN {X 0,Y 560.271,Z 395.943,A -85,B 0,C 180,E1 26629.304,E2 26629.304} C_VEL
LIN {X 0,Y 560.262,Z 395.941,A -85,B 0,C 180,E1 26626.059,E2 26626.059} C_VEL
LIN {X 0,Y 560.269,Z 395.94,A -85,B 0,C 180,E1 26622.768,E2 26622.768} C_VEL
LIN {X 0,Y 560.27,Z 395.946,A -85,B 0,C 180,E1 26619.417,E2 26619.417} C_VEL
LIN {X 0,Y 560.268,Z 395.939,A -85,B 0,C 180,E1 26615.991,E2 26615.991} C_VEL
LIN {X 0,Y 560.273,Z 395.944,A -85,B 0,C 180,E1 26612.701,E2 26612.701} C_VEL
LIN {X 0,Y 560.258,Z 395.944,A -85,B 0,C 180,E1 26609.428,E2 26609.428} C_VEL
LIN {X 0,Y 560.275,Z 395.941,A -85,B 0,C 180,E1 26606.083,E2 26606.083} C_VEL
LIN {X 0,Y 560.271,Z 395.948,A -85,B 0,C 180,E1 26602.744,E2 26602.744} C_VEL
LIN {X 0,Y 560.262,Z 395.939,A -85,B 0,C 180,E1 26599.33,E2 26599.33} C_VEL
LIN {X 0,Y 560.27,Z 395.93,A -85,B 0,C 180,E1 26595.989,E2 26595.989} C_VEL
LIN {X 0,Y 560.255,Z 395.938,A -85,B 0,C 180,E1 26592.702,E2 26592.702} C_VEL
LIN {X 0,Y 560.315,Z 396.2,A -85,B 0,C 180,E1 26589.474,E2 26589.474} C_VEL
LIN {X 0,Y 561.644,Z 399.522,A -85,B 0,C 180,E1 26589.088,E2 26589.088} C_VEL
LIN {X 0,Y 567.247,Z 412.43,A -85,B 0,C 180,E1 26587.773,E2 26587.773} C_VEL
LIN {X 0,Y 566.402,Z 455.666,A -85,B 0,C 180,E1 26585.067,E2 26585.067} C_VEL
LIN {X 0,Y 567.762,Z 464.856,A -85,B 0,C 180,E1 26584.831,E2 26584.831} C_VEL
LIN {X 0,Y 566.434,Z 684.991,A -85,B 0,C 180,E1 26581.653,E2 26581.653} C_VEL
LIN {X 0,Y 565.939,Z 762.176,A -85,B 0,C 180,E1 26580.53,E2 26580.53} C_VEL
LIN {X 0,Y 565.546,Z 783.591,A -85,B 0,C 180,E1 26580.027,E2 26580.027} C_VEL
LIN {X 0,Y 565.084,Z 805.523,A -85,B 0,C 180,E1 26579.318,E2 26579.318} C_VEL
LIN {X 0,Y 564.576,Z 826.359,A -85,B 0,C 180,E1 26578.452,E2 26578.452} C_VEL
LIN {X 0,Y 563.945,Z 846.462,A -85,B 0,C 180,E1 26577.409,E2 26577.409} C_VEL
LIN {X 0,Y 563.333,Z 866.312,A -85,B 0,C 180,E1 26576.173,E2 26576.173} C_VEL
LIN {X 0,Y 562.708,Z 885.096,A -85,B 0,C 180,E1 26574.795,E2 26574.795} C_VEL
LIN {X 0,Y 562.112,Z 902.883,A -85,B 0,C 180,E1 26573.26,E2 26573.26} C_VEL
LIN {X 0,Y 561.591,Z 919.164,A -85,B 0,C 180,E1 26571.627,E2 26571.627} C_VEL
LIN {X 0,Y 561.112,Z 935.007,A -85,B 0,C 180,E1 26569.791,E2 26569.791} C_VEL
LIN {X 0,Y 560.744,Z 948.616,A -85,B 0,C 180,E1 26567.969,E2 26567.969} C_VEL
LIN {X 0,Y 560.423,Z 961.456,A -85,B 0,C 180,E1 26565.949,E2 26565.949} C_VEL
LIN {X 0,Y 560.212,Z 972.284,A -85,B 0,C 180,E1 26563.944,E2 26563.944} C_VEL
LIN {X 0,Y 560.068,Z 981.838,A -85,B 0,C 180,E1 26561.849,E2 26561.849} C_VEL
LIN {X 0,Y 559.973,Z 989.524,A -85,B 0,C 180,E1 26559.768,E2 26559.768} C_VEL
LIN {X 0,Y 559.927,Z 995.886,A -85,B 0,C 180,E1 26557.595,E2 26557.595} C_VEL
LIN {X 0,Y 559.918,Z 1000.423,A -85,B 0,C 180,E1 26555.536,E2 26555.536} C_VEL
LIN {X 0,Y 559.915,Z 1003.558,A -85,B 0,C 180,E1 26553.38,E2 26553.38} C_VEL
LIN {X 0,Y 559.913,Z 1005.261,A -85,B 0,C 180,E1 26551.128,E2 26551.128} C_VEL
LIN {X 0,Y 559.907,Z 1005.284,A -85,B 0,C 180,E1 26548.979,E2 26548.979} C_VEL
LIN {X 0,Y 559.91,Z 1003.674,A -85,B 0,C 180,E1 26546.726,E2 26546.726} C_VEL
LIN {X 0,Y 559.911,Z 1000.636,A -85,B 0,C 180,E1 26544.572,E2 26544.572} C_VEL
